ABB RAPID module: P85.mod

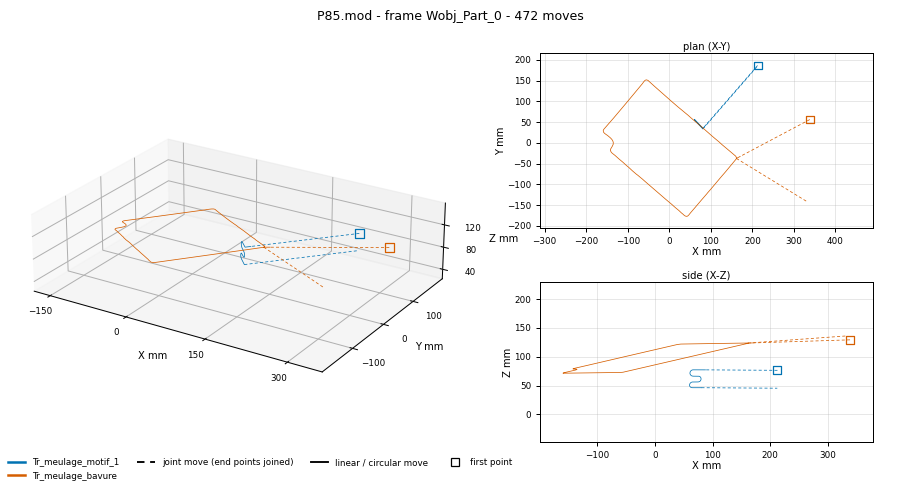
[picture p0: tool path of P85.mod in frame Wobj_Part_0, 472 of 479 moves have a stored position in this frame; points joined in program order, loops and branches not executed]
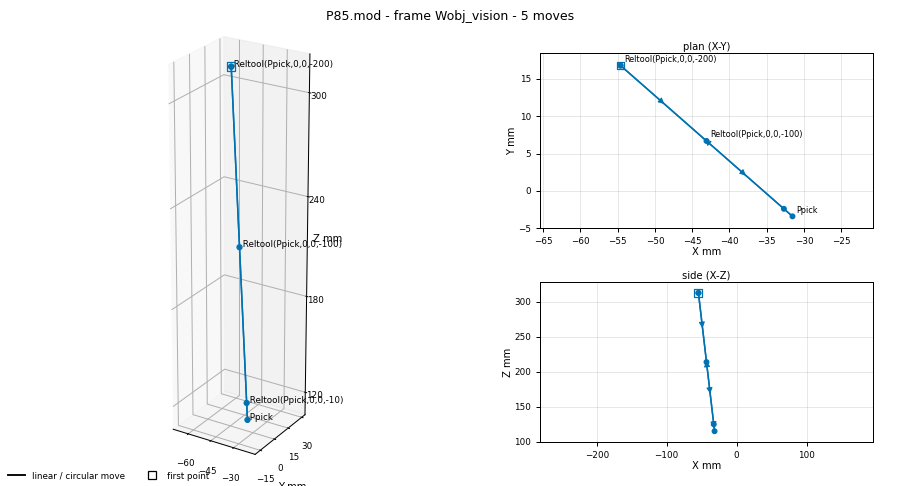
[picture p1: tool path of P85.mod in frame Wobj_vision, 5 of 479 moves have a stored position in this frame; points joined in program order, loops and branches not executed]
MODULE P85
	LOCAL CONST Speeddata vitesse_Tronconnage :=[10, 500, 0, 0];
	LOCAL CONST Robtarget Tr_meulage_motif_1_App1 :=[[212.414841209805,186.150509126283,76.4688798702914],[0.248270770432822,-0.247228008216849,-0.660888683117367,0.663676189891738],[0,0,0,0],[8.999999E+09,8.999999E+09,8.999999E+09,8.999999E+09,8.999999E+09,8.999999E+09]];
	LOCAL CONST Robtarget Tr_meulage_motif_1_App2 :=[[87.7145408886153,42.8006029953767,77.2685748528896],[0.248270770432822,-0.247228008216849,-0.660888683117367,0.663676189891738],[0,0,0,0],[8.999999E+09,8.999999E+09,8.999999E+09,8.999999E+09,8.999999E+09,8.999999E+09]];
	LOCAL CONST Robtarget Tr_meulage_motif_1_P0 :=[[81.1513671875,35.25587109375,77.3106640625],[0.248270770432822,-0.247228008216849,-0.660888683117367,0.663676189891738],[0,0,0,0],[8.999999E+09,8.999999E+09,8.999999E+09,8.999999E+09,8.999999E+09,8.999999E+09]];
	LOCAL CONST Robtarget Tr_meulage_motif_1_P1 :=[[80.4589453125,35.97736328125,77.3106875],[0.248270770432822,-0.247228008216849,-0.660888683117367,0.663676189891738],[0,0,0,0],[8.999999E+09,8.999999E+09,8.999999E+09,8.999999E+09,8.999999E+09,8.999999E+09]];
	LOCAL CONST Robtarget Tr_meulage_motif_1_P2 :=[[79.7665234375,36.69885546875,77.310703125],[0.248270770432822,-0.247228008216849,-0.660888683117367,0.663676189891738],[0,0,0,0],[8.999999E+09,8.999999E+09,8.999999E+09,8.999999E+09,8.999999E+09,8.999999E+09]];
	LOCAL CONST Robtarget Tr_meulage_motif_1_P3 :=[[79.0741015625,37.4203515625,77.3107265625],[0.248270770432822,-0.247228008216849,-0.660888683117367,0.663676189891738],[0,0,0,0],[8.999999E+09,8.999999E+09,8.999999E+09,8.999999E+09,8.999999E+09,8.999999E+09]];
	LOCAL CONST Robtarget Tr_meulage_motif_1_P4 :=[[78.3816796875,38.14184375,77.3107421875],[0.248270770432822,-0.247228008216849,-0.660888683117367,0.663676189891738],[0,0,0,0],[8.999999E+09,8.999999E+09,8.999999E+09,8.999999E+09,8.999999E+09,8.999999E+09]];
	LOCAL CONST Robtarget Tr_meulage_motif_1_P5 :=[[77.6892578125,38.8633359375,77.3107578125],[0.248270770432822,-0.247228008216849,-0.660888683117367,0.663676189891738],[0,0,0,0],[8.999999E+09,8.999999E+09,8.999999E+09,8.999999E+09,8.999999E+09,8.999999E+09]];
	LOCAL CONST Robtarget Tr_meulage_motif_1_P6 :=[[76.9968359375,39.584828125,77.31078125],[0.248270770432822,-0.247228008216849,-0.660888683117367,0.663676189891738],[0,0,0,0],[8.999999E+09,8.999999E+09,8.999999E+09,8.999999E+09,8.999999E+09,8.999999E+09]];
	LOCAL CONST Robtarget Tr_meulage_motif_1_P7 :=[[76.3044140625,40.3063203125,77.310796875],[0.248270770432822,-0.247228008216849,-0.660888683117367,0.663676189891738],[0,0,0,0],[8.999999E+09,8.999999E+09,8.999999E+09,8.999999E+09,8.999999E+09,8.999999E+09]];
	LOCAL CONST Robtarget Tr_meulage_motif_1_P8 :=[[75.6119921875,41.0278125,77.3108203125],[0.248270770432822,-0.247228008216849,-0.660888683117367,0.663676189891738],[0,0,0,0],[8.999999E+09,8.999999E+09,8.999999E+09,8.999999E+09,8.999999E+09,8.999999E+09]];
	LOCAL CONST Robtarget Tr_meulage_motif_1_P9 :=[[74.9195703125,41.7493046875,77.3108359375],[0.248270770432822,-0.247228008216849,-0.660888683117367,0.663676189891738],[0,0,0,0],[8.999999E+09,8.999999E+09,8.999999E+09,8.999999E+09,8.999999E+09,8.999999E+09]];
	LOCAL CONST Robtarget Tr_meulage_motif_1_P10 :=[[74.2271484375,42.47080078125,77.310859375],[0.248270770432822,-0.247228008216849,-0.660888683117367,0.663676189891738],[0,0,0,0],[8.999999E+09,8.999999E+09,8.999999E+09,8.999999E+09,8.999999E+09,8.999999E+09]];
	LOCAL CONST Robtarget Tr_meulage_motif_1_P11 :=[[73.5347265625,43.19229296875,77.310875],[0.248270770432822,-0.247228008216849,-0.660888683117367,0.663676189891738],[0,0,0,0],[8.999999E+09,8.999999E+09,8.999999E+09,8.999999E+09,8.999999E+09,8.999999E+09]];
	LOCAL CONST Robtarget Tr_meulage_motif_1_P12 :=[[72.8423046875,43.91378515625,77.310890625],[0.248270770432822,-0.247228008216849,-0.660888683117367,0.663676189891738],[0,0,0,0],[8.999999E+09,8.999999E+09,8.999999E+09,8.999999E+09,8.999999E+09,8.999999E+09]];
	LOCAL CONST Robtarget Tr_meulage_motif_1_P13 :=[[72.1498828125,44.63527734375,77.3109140625],[0.248270770432822,-0.247228008216849,-0.660888683117367,0.663676189891738],[0,0,0,0],[8.999999E+09,8.999999E+09,8.999999E+09,8.999999E+09,8.999999E+09,8.999999E+09]];
	LOCAL CONST Robtarget Tr_meulage_motif_1_P14 :=[[71.4574609375,45.35676953125,77.3109296875],[0.248270770432822,-0.247228008216849,-0.660888683117367,0.663676189891738],[0,0,0,0],[8.999999E+09,8.999999E+09,8.999999E+09,8.999999E+09,8.999999E+09,8.999999E+09]];
	LOCAL CONST Robtarget Tr_meulage_motif_1_P15 :=[[70.7650390625,46.07826171875,77.310953125],[0.248270770432822,-0.247228008216849,-0.660888683117367,0.663676189891738],[0,0,0,0],[8.999999E+09,8.999999E+09,8.999999E+09,8.999999E+09,8.999999E+09,8.999999E+09]];
	LOCAL CONST Robtarget Tr_meulage_motif_1_P16 :=[[70.0726171875,46.79975390625,77.31096875],[0.248270770432822,-0.247228008216849,-0.660888683117367,0.663676189891738],[0,0,0,0],[8.999999E+09,8.999999E+09,8.999999E+09,8.999999E+09,8.999999E+09,8.999999E+09]];
	LOCAL CONST Robtarget Tr_meulage_motif_1_P17 :=[[69.3801953125,47.52125,77.310984375],[0.248270770432822,-0.247228008216849,-0.660888683117367,0.663676189891738],[0,0,0,0],[8.999999E+09,8.999999E+09,8.999999E+09,8.999999E+09,8.999999E+09,8.999999E+09]];
	LOCAL CONST Robtarget Tr_meulage_motif_1_P18 :=[[68.6877734375,48.2427421875,77.3110078125],[0.248270770432822,-0.247228008216849,-0.660888683117367,0.663676189891738],[0,0,0,0],[8.999999E+09,8.999999E+09,8.999999E+09,8.999999E+09,8.999999E+09,8.999999E+09]];
	LOCAL CONST Robtarget Tr_meulage_motif_1_P19 :=[[67.9953515625,48.964234375,77.3110234375],[0.248270770432822,-0.247228008216849,-0.660888683117367,0.663676189891738],[0,0,0,0],[8.999999E+09,8.999999E+09,8.999999E+09,8.999999E+09,8.999999E+09,8.999999E+09]];
	LOCAL CONST Robtarget Tr_meulage_motif_1_P20 :=[[67.3029296875,49.6857265625,77.311046875],[0.248270770432822,-0.247228008216849,-0.660888683117367,0.663676189891738],[0,0,0,0],[8.999999E+09,8.999999E+09,8.999999E+09,8.999999E+09,8.999999E+09,8.999999E+09]];
	LOCAL CONST Robtarget Tr_meulage_motif_1_P21 :=[[66.6105078125,50.40721875,77.3110625],[0.248270770432822,-0.247228008216849,-0.660888683117367,0.663676189891738],[0,0,0,0],[8.999999E+09,8.999999E+09,8.999999E+09,8.999999E+09,8.999999E+09,8.999999E+09]];
	LOCAL CONST Robtarget Tr_meulage_motif_1_P22 :=[[65.9180859375,51.1287109375,77.3110859375],[0.248270770432822,-0.247228008216849,-0.660888683117367,0.663676189891738],[0,0,0,0],[8.999999E+09,8.999999E+09,8.999999E+09,8.999999E+09,8.999999E+09,8.999999E+09]];
	LOCAL CONST Robtarget Tr_meulage_motif_1_P23 :=[[65.22724609375,51.84141796875,77.2006171875],[0.248270770432822,-0.247228008216849,-0.660888683117367,0.663676189891738],[0,0,0,0],[8.999999E+09,8.999999E+09,8.999999E+09,8.999999E+09,8.999999E+09,8.999999E+09]];
	LOCAL CONST Robtarget Tr_meulage_motif_1_P24 :=[[64.56505859375,52.51778515625,76.98965625],[0.248270770432822,-0.247228008216849,-0.660888683117367,0.663676189891738],[0,0,0,0],[8.999999E+09,8.999999E+09,8.999999E+09,8.999999E+09,8.999999E+09,8.999999E+09]];
	LOCAL CONST Robtarget Tr_meulage_motif_1_P25 :=[[63.96585546875,53.124609375,76.7181015625],[0.248270770432822,-0.247228008216849,-0.660888683117367,0.663676189891738],[0,0,0,0],[8.999999E+09,8.999999E+09,8.999999E+09,8.999999E+09,8.999999E+09,8.999999E+09]];
	LOCAL CONST Robtarget Tr_meulage_motif_1_P26 :=[[63.43768359375,53.65715234375,76.442453125],[0.248270770432822,-0.247228008216849,-0.660888683117367,0.663676189891738],[0,0,0,0],[8.999999E+09,8.999999E+09,8.999999E+09,8.999999E+09,8.999999E+09,8.999999E+09]];
	LOCAL CONST Robtarget Tr_meulage_motif_1_P27 :=[[62.655421875,54.432515625,75.82696875],[0.248270770432822,-0.247228008216849,-0.660888683117367,0.663676189891738],[0,0,0,0],[8.999999E+09,8.999999E+09,8.999999E+09,8.999999E+09,8.999999E+09,8.999999E+09]];
	LOCAL CONST Robtarget Tr_meulage_motif_1_P28 :=[[61.91913671875,55.14502734375,74.980171875],[0.248270770432822,-0.247228008216849,-0.660888683117367,0.663676189891738],[0,0,0,0],[8.999999E+09,8.999999E+09,8.999999E+09,8.999999E+09,8.999999E+09,8.999999E+09]];
	LOCAL CONST Robtarget Tr_meulage_motif_1_P29 :=[[61.29919140625,55.724953125,73.9573359375],[0.248270770432822,-0.247228008216849,-0.660888683117367,0.663676189891738],[0,0,0,0],[8.999999E+09,8.999999E+09,8.999999E+09,8.999999E+09,8.999999E+09,8.999999E+09]];
	LOCAL CONST Robtarget Tr_meulage_motif_1_P30 :=[[60.9251953125,56.04264453125,72.8422734375],[0.248270770432822,-0.247228008216849,-0.660888683117367,0.663676189891738],[0,0,0,0],[8.999999E+09,8.999999E+09,8.999999E+09,8.999999E+09,8.999999E+09,8.999999E+09]];
	LOCAL CONST Robtarget Tr_meulage_motif_1_P31 :=[[60.884015625,56.04065625,72.147],[0.248270770432822,-0.247228008216849,-0.660888683117367,0.663676189891738],[0,0,0,0],[8.999999E+09,8.999999E+09,8.999999E+09,8.999999E+09,8.999999E+09,8.999999E+09]];
	LOCAL CONST Robtarget Tr_meulage_motif_1_P32 :=[[60.86269921875,56.0202109375,71.4864140625],[0.248270770432822,-0.247228008216849,-0.660888683117367,0.663676189891738],[0,0,0,0],[8.999999E+09,8.999999E+09,8.999999E+09,8.999999E+09,8.999999E+09,8.999999E+09]];
	LOCAL CONST Robtarget Tr_meulage_motif_1_P33 :=[[60.87937890625,55.9601796875,70.8259765625],[0.248270770432822,-0.247228008216849,-0.660888683117367,0.663676189891738],[0,0,0,0],[8.999999E+09,8.999999E+09,8.999999E+09,8.999999E+09,8.999999E+09,8.999999E+09]];
	LOCAL CONST Robtarget Tr_meulage_motif_1_P34 :=[[61.1888359375,55.56666015625,69.7253125],[0.248270770432822,-0.247228008216849,-0.660888683117367,0.663676189891738],[0,0,0,0],[8.999999E+09,8.999999E+09,8.999999E+09,8.999999E+09,8.999999E+09,8.999999E+09]];
	LOCAL CONST Robtarget Tr_meulage_motif_1_P35 :=[[61.74952734375,54.9174921875,68.7196796875],[0.248270770432822,-0.247228008216849,-0.660888683117367,0.663676189891738],[0,0,0,0],[8.999999E+09,8.999999E+09,8.999999E+09,8.999999E+09,8.999999E+09,8.999999E+09]];
	LOCAL CONST Robtarget Tr_meulage_motif_1_P36 :=[[62.43143359375,54.153484375,67.891609375],[0.248270770432822,-0.247228008216849,-0.660888683117367,0.663676189891738],[0,0,0,0],[8.999999E+09,8.999999E+09,8.999999E+09,8.999999E+09,8.999999E+09,8.999999E+09]];
	LOCAL CONST Robtarget Tr_meulage_motif_1_P37 :=[[62.89443359375,53.645515625,67.4962421875],[0.248270770432822,-0.247228008216849,-0.660888683117367,0.663676189891738],[0,0,0,0],[8.999999E+09,8.999999E+09,8.999999E+09,8.999999E+09,8.999999E+09,8.999999E+09]];
	LOCAL CONST Robtarget Tr_meulage_motif_1_P38 :=[[63.6806484375,52.79484375,67.0091796875],[0.248270770432822,-0.247228008216849,-0.660888683117367,0.663676189891738],[0,0,0,0],[8.999999E+09,8.999999E+09,8.999999E+09,8.999999E+09,8.999999E+09,8.999999E+09]];
	LOCAL CONST Robtarget Tr_meulage_motif_1_P39 :=[[64.25725390625,52.17699609375,66.745328125],[0.248270770432822,-0.247228008216849,-0.660888683117367,0.663676189891738],[0,0,0,0],[8.999999E+09,8.999999E+09,8.999999E+09,8.999999E+09,8.999999E+09,8.999999E+09]];
	LOCAL CONST Robtarget Tr_meulage_motif_1_P40 :=[[64.89599609375,51.4982421875,66.541046875],[0.248270770432822,-0.247228008216849,-0.660888683117367,0.663676189891738],[0,0,0,0],[8.999999E+09,8.999999E+09,8.999999E+09,8.999999E+09,8.999999E+09,8.999999E+09]];
	LOCAL CONST Robtarget Tr_meulage_motif_1_P41 :=[[65.5721484375,50.7866953125,66.432546875],[0.248270770432822,-0.247228008216849,-0.660888683117367,0.663676189891738],[0,0,0,0],[8.999999E+09,8.999999E+09,8.999999E+09,8.999999E+09,8.999999E+09,8.999999E+09]];
	LOCAL CONST Robtarget Tr_meulage_motif_1_P42 :=[[66.255859375,50.0671484375,66.3220390625],[0.248270770432822,-0.247228008216849,-0.660888683117367,0.663676189891738],[0,0,0,0],[8.999999E+09,8.999999E+09,8.999999E+09,8.999999E+09,8.999999E+09,8.999999E+09]];
	LOCAL CONST Robtarget Tr_meulage_motif_1_P43 :=[[66.94828125,49.34565625,66.3220234375],[0.248270770432822,-0.247228008216849,-0.660888683117367,0.663676189891738],[0,0,0,0],[8.999999E+09,8.999999E+09,8.999999E+09,8.999999E+09,8.999999E+09,8.999999E+09]];
	LOCAL CONST Robtarget Tr_meulage_motif_1_P44 :=[[67.640703125,48.6241640625,66.3220078125],[0.248270770432822,-0.247228008216849,-0.660888683117367,0.663676189891738],[0,0,0,0],[8.999999E+09,8.999999E+09,8.999999E+09,8.999999E+09,8.999999E+09,8.999999E+09]];
	LOCAL CONST Robtarget Tr_meulage_motif_1_P45 :=[[68.333125,47.902671875,66.321984375],[0.248270770432822,-0.247228008216849,-0.660888683117367,0.663676189891738],[0,0,0,0],[8.999999E+09,8.999999E+09,8.999999E+09,8.999999E+09,8.999999E+09,8.999999E+09]];
	LOCAL CONST Robtarget Tr_meulage_motif_1_P46 :=[[69.025546875,47.1811796875,66.32196875],[0.248270770432822,-0.247228008216849,-0.660888683117367,0.663676189891738],[0,0,0,0],[8.999999E+09,8.999999E+09,8.999999E+09,8.999999E+09,8.999999E+09,8.999999E+09]];
	LOCAL CONST Robtarget Tr_meulage_motif_1_P47 :=[[69.71796875,46.4596875,66.3219453125],[0.248270770432822,-0.247228008216849,-0.660888683117367,0.663676189891738],[0,0,0,0],[8.999999E+09,8.999999E+09,8.999999E+09,8.999999E+09,8.999999E+09,8.999999E+09]];
	LOCAL CONST Robtarget Tr_meulage_motif_1_P48 :=[[70.410390625,45.73819140625,66.3219296875],[0.248270770432822,-0.247228008216849,-0.660888683117367,0.663676189891738],[0,0,0,0],[8.999999E+09,8.999999E+09,8.999999E+09,8.999999E+09,8.999999E+09,8.999999E+09]];
	LOCAL CONST Robtarget Tr_meulage_motif_1_P49 :=[[71.1028125,45.01669921875,66.3219140625],[0.248270770432822,-0.247228008216849,-0.660888683117367,0.663676189891738],[0,0,0,0],[8.999999E+09,8.999999E+09,8.999999E+09,8.999999E+09,8.999999E+09,8.999999E+09]];
	LOCAL CONST Robtarget Tr_meulage_motif_1_P50 :=[[71.795234375,44.29520703125,66.321890625],[0.248270770432822,-0.247228008216849,-0.660888683117367,0.663676189891738],[0,0,0,0],[8.999999E+09,8.999999E+09,8.999999E+09,8.999999E+09,8.999999E+09,8.999999E+09]];
	LOCAL CONST Robtarget Tr_meulage_motif_1_P51 :=[[72.48765625,43.57371484375,66.321875],[0.248270770432822,-0.247228008216849,-0.660888683117367,0.663676189891738],[0,0,0,0],[8.999999E+09,8.999999E+09,8.999999E+09,8.999999E+09,8.999999E+09,8.999999E+09]];
	LOCAL CONST Robtarget Tr_meulage_motif_1_P52 :=[[73.180078125,42.85222265625,66.3218515625],[0.248270770432822,-0.247228008216849,-0.660888683117367,0.663676189891738],[0,0,0,0],[8.999999E+09,8.999999E+09,8.999999E+09,8.999999E+09,8.999999E+09,8.999999E+09]];
	LOCAL CONST Robtarget Tr_meulage_motif_1_P53 :=[[73.8725,42.13073046875,66.3218359375],[0.248270770432822,-0.247228008216849,-0.660888683117367,0.663676189891738],[0,0,0,0],[8.999999E+09,8.999999E+09,8.999999E+09,8.999999E+09,8.999999E+09,8.999999E+09]];
	LOCAL CONST Robtarget Tr_meulage_motif_1_P54 :=[[74.564921875,41.40923828125,66.3218125],[0.248270770432822,-0.247228008216849,-0.660888683117367,0.663676189891738],[0,0,0,0],[8.999999E+09,8.999999E+09,8.999999E+09,8.999999E+09,8.999999E+09,8.999999E+09]];
	LOCAL CONST Robtarget Tr_meulage_motif_1_P55 :=[[75.25734375,40.6877421875,66.321796875],[0.248270770432822,-0.247228008216849,-0.660888683117367,0.663676189891738],[0,0,0,0],[8.999999E+09,8.999999E+09,8.999999E+09,8.999999E+09,8.999999E+09,8.999999E+09]];
	LOCAL CONST Robtarget Tr_meulage_motif_1_P56 :=[[75.949765625,39.96625,66.32178125],[0.248270770432822,-0.247228008216849,-0.660888683117367,0.663676189891738],[0,0,0,0],[8.999999E+09,8.999999E+09,8.999999E+09,8.999999E+09,8.999999E+09,8.999999E+09]];
	LOCAL CONST Robtarget Tr_meulage_motif_1_P57 :=[[76.63346875,39.24670703125,66.2112734375],[0.248270770432822,-0.247228008216849,-0.660888683117367,0.663676189891738],[0,0,0,0],[8.999999E+09,8.999999E+09,8.999999E+09,8.999999E+09,8.999999E+09,8.999999E+09]];
	LOCAL CONST Robtarget Tr_meulage_motif_1_P58 :=[[77.2820390625,38.55728515625,66.00028125],[0.248270770432822,-0.247228008216849,-0.660888683117367,0.663676189891738],[0,0,0,0],[8.999999E+09,8.999999E+09,8.999999E+09,8.999999E+09,8.999999E+09,8.999999E+09]];
	LOCAL CONST Robtarget Tr_meulage_motif_1_P59 :=[[77.86371875,37.9336484375,65.7286953125],[0.248270770432822,-0.247228008216849,-0.660888683117367,0.663676189891738],[0,0,0,0],[8.999999E+09,8.999999E+09,8.999999E+09,8.999999E+09,8.999999E+09,8.999999E+09]];
	LOCAL CONST Robtarget Tr_meulage_motif_1_P60 :=[[78.3465703125,37.41090234375,65.424828125],[0.248270770432822,-0.247228008216849,-0.660888683117367,0.663676189891738],[0,0,0,0],[8.999999E+09,8.999999E+09,8.999999E+09,8.999999E+09,8.999999E+09,8.999999E+09]];
	LOCAL CONST Robtarget Tr_meulage_motif_1_P61 :=[[79.0415,36.64405859375,64.7629375],[0.248270770432822,-0.247228008216849,-0.660888683117367,0.663676189891738],[0,0,0,0],[8.999999E+09,8.999999E+09,8.999999E+09,8.999999E+09,8.999999E+09,8.999999E+09]];
	LOCAL CONST Robtarget Tr_meulage_motif_1_P62 :=[[79.6369375,35.96543359375,63.8618828125],[0.248270770432822,-0.247228008216849,-0.660888683117367,0.663676189891738],[0,0,0,0],[8.999999E+09,8.999999E+09,8.999999E+09,8.999999E+09,8.999999E+09,8.999999E+09]];
	LOCAL CONST Robtarget Tr_meulage_motif_1_P63 :=[[79.973640625,35.54712109375,62.81688671875],[0.248270770432822,-0.247228008216849,-0.660888683117367,0.663676189891738],[0,0,0,0],[8.999999E+09,8.999999E+09,8.999999E+09,8.999999E+09,8.999999E+09,8.999999E+09]];
	LOCAL CONST Robtarget Tr_meulage_motif_1_P64 :=[[80.079234375,35.39237109375,62.12435546875],[0.248270770432822,-0.247228008216849,-0.660888683117367,0.663676189891738],[0,0,0,0],[8.999999E+09,8.999999E+09,8.999999E+09,8.999999E+09,8.999999E+09,8.999999E+09]];
	LOCAL CONST Robtarget Tr_meulage_motif_1_P65 :=[[80.0986171875,35.32250390625,61.35512109375],[0.248270770432822,-0.247228008216849,-0.660888683117367,0.663676189891738],[0,0,0,0],[8.999999E+09,8.999999E+09,8.999999E+09,8.999999E+09,8.999999E+09,8.999999E+09]];
	LOCAL CONST Robtarget Tr_meulage_motif_1_P66 :=[[80.0274453125,35.34699609375,60.586015625],[0.248270770432822,-0.247228008216849,-0.660888683117367,0.663676189891738],[0,0,0,0],[8.999999E+09,8.999999E+09,8.999999E+09,8.999999E+09,8.999999E+09,8.999999E+09]];
	LOCAL CONST Robtarget Tr_meulage_motif_1_P67 :=[[79.7011796875,35.61546875,59.4788828125],[0.248270770432822,-0.247228008216849,-0.660888683117367,0.663676189891738],[0,0,0,0],[8.999999E+09,8.999999E+09,8.999999E+09,8.999999E+09,8.999999E+09,8.999999E+09]];
	LOCAL CONST Robtarget Tr_meulage_motif_1_P68 :=[[79.395421875,35.89628515625,58.89378515625],[0.248270770432822,-0.247228008216849,-0.660888683117367,0.663676189891738],[0,0,0,0],[8.999999E+09,8.999999E+09,8.999999E+09,8.999999E+09,8.999999E+09,8.999999E+09]];
	LOCAL CONST Robtarget Tr_meulage_motif_1_P69 :=[[78.7525546875,36.5089140625,58.0075625],[0.248270770432822,-0.247228008216849,-0.660888683117367,0.663676189891738],[0,0,0,0],[8.999999E+09,8.999999E+09,8.999999E+09,8.999999E+09,8.999999E+09,8.999999E+09]];
	LOCAL CONST Robtarget Tr_meulage_motif_1_P70 :=[[78.3336484375,36.91867578125,57.59367578125],[0.248270770432822,-0.247228008216849,-0.660888683117367,0.663676189891738],[0,0,0,0],[8.999999E+09,8.999999E+09,8.999999E+09,8.999999E+09,8.999999E+09,8.999999E+09]];
	LOCAL CONST Robtarget Tr_meulage_motif_1_P71 :=[[77.542046875,37.7084140625,57.05014453125],[0.248270770432822,-0.247228008216849,-0.660888683117367,0.663676189891738],[0,0,0,0],[8.999999E+09,8.999999E+09,8.999999E+09,8.999999E+09,8.999999E+09,8.999999E+09]];
	LOCAL CONST Robtarget Tr_meulage_motif_1_P72 :=[[76.960859375,38.2949375,56.75495703125],[0.248270770432822,-0.247228008216849,-0.660888683117367,0.663676189891738],[0,0,0,0],[8.999999E+09,8.999999E+09,8.999999E+09,8.999999E+09,8.999999E+09,8.999999E+09]];
	LOCAL CONST Robtarget Tr_meulage_motif_1_P73 :=[[76.3089296875,38.961046875,56.5507109375],[0.248270770432822,-0.247228008216849,-0.660888683117367,0.663676189891738],[0,0,0,0],[8.999999E+09,8.999999E+09,8.999999E+09,8.999999E+09,8.999999E+09,8.999999E+09]];
	LOCAL CONST Robtarget Tr_meulage_motif_1_P74 :=[[75.6257734375,39.6658828125,56.4422421875],[0.248270770432822,-0.247228008216849,-0.660888683117367,0.663676189891738],[0,0,0,0],[8.999999E+09,8.999999E+09,8.999999E+09,8.999999E+09,8.999999E+09,8.999999E+09]];
	LOCAL CONST Robtarget Tr_meulage_motif_1_P75 :=[[74.9349375,40.37858984375,56.33177734375],[0.248270770432822,-0.247228008216849,-0.660888683117367,0.663676189891738],[0,0,0,0],[8.999999E+09,8.999999E+09,8.999999E+09,8.999999E+09,8.999999E+09,8.999999E+09]];
	LOCAL CONST Robtarget Tr_meulage_motif_1_P76 :=[[74.242515625,41.10008203125,56.331796875],[0.248270770432822,-0.247228008216849,-0.660888683117367,0.663676189891738],[0,0,0,0],[8.999999E+09,8.999999E+09,8.999999E+09,8.999999E+09,8.999999E+09,8.999999E+09]];
	LOCAL CONST Robtarget Tr_meulage_motif_1_P77 :=[[73.55009375,41.82157421875,56.33181640625],[0.248270770432822,-0.247228008216849,-0.660888683117367,0.663676189891738],[0,0,0,0],[8.999999E+09,8.999999E+09,8.999999E+09,8.999999E+09,8.999999E+09,8.999999E+09]];
	LOCAL CONST Robtarget Tr_meulage_motif_1_P78 :=[[72.857671875,42.54306640625,56.3318359375],[0.248270770432822,-0.247228008216849,-0.660888683117367,0.663676189891738],[0,0,0,0],[8.999999E+09,8.999999E+09,8.999999E+09,8.999999E+09,8.999999E+09,8.999999E+09]];
	LOCAL CONST Robtarget Tr_meulage_motif_1_P79 :=[[72.16525,43.26455859375,56.33185546875],[0.248270770432822,-0.247228008216849,-0.660888683117367,0.663676189891738],[0,0,0,0],[8.999999E+09,8.999999E+09,8.999999E+09,8.999999E+09,8.999999E+09,8.999999E+09]];
	LOCAL CONST Robtarget Tr_meulage_motif_1_P80 :=[[71.472828125,43.9860546875,56.33187109375],[0.248270770432822,-0.247228008216849,-0.660888683117367,0.663676189891738],[0,0,0,0],[8.999999E+09,8.999999E+09,8.999999E+09,8.999999E+09,8.999999E+09,8.999999E+09]];
	LOCAL CONST Robtarget Tr_meulage_motif_1_P81 :=[[70.78040625,44.707546875,56.331890625],[0.248270770432822,-0.247228008216849,-0.660888683117367,0.663676189891738],[0,0,0,0],[8.999999E+09,8.999999E+09,8.999999E+09,8.999999E+09,8.999999E+09,8.999999E+09]];
	LOCAL CONST Robtarget Tr_meulage_motif_1_P82 :=[[70.087984375,45.4290390625,56.33191015625],[0.248270770432822,-0.247228008216849,-0.660888683117367,0.663676189891738],[0,0,0,0],[8.999999E+09,8.999999E+09,8.999999E+09,8.999999E+09,8.999999E+09,8.999999E+09]];
	LOCAL CONST Robtarget Tr_meulage_motif_1_P83 :=[[69.3955625,46.15053125,56.3319296875],[0.248270770432822,-0.247228008216849,-0.660888683117367,0.663676189891738],[0,0,0,0],[8.999999E+09,8.999999E+09,8.999999E+09,8.999999E+09,8.999999E+09,8.999999E+09]];
	LOCAL CONST Robtarget Tr_meulage_motif_1_P84 :=[[68.703140625,46.8720234375,56.33194921875],[0.248270770432822,-0.247228008216849,-0.660888683117367,0.663676189891738],[0,0,0,0],[8.999999E+09,8.999999E+09,8.999999E+09,8.999999E+09,8.999999E+09,8.999999E+09]];
	LOCAL CONST Robtarget Tr_meulage_motif_1_P85 :=[[68.01071875,47.593515625,56.33196875],[0.248270770432822,-0.247228008216849,-0.660888683117367,0.663676189891738],[0,0,0,0],[8.999999E+09,8.999999E+09,8.999999E+09,8.999999E+09,8.999999E+09,8.999999E+09]];
	LOCAL CONST Robtarget Tr_meulage_motif_1_P86 :=[[67.318296875,48.3150078125,56.331984375],[0.248270770432822,-0.247228008216849,-0.660888683117367,0.663676189891738],[0,0,0,0],[8.999999E+09,8.999999E+09,8.999999E+09,8.999999E+09,8.999999E+09,8.999999E+09]];
	LOCAL CONST Robtarget Tr_meulage_motif_1_P87 :=[[66.625875,49.03650390625,56.33200390625],[0.248270770432822,-0.247228008216849,-0.660888683117367,0.663676189891738],[0,0,0,0],[8.999999E+09,8.999999E+09,8.999999E+09,8.999999E+09,8.999999E+09,8.999999E+09]];
	LOCAL CONST Robtarget Tr_meulage_motif_1_P88 :=[[65.933453125,49.75799609375,56.3320234375],[0.248270770432822,-0.247228008216849,-0.660888683117367,0.663676189891738],[0,0,0,0],[8.999999E+09,8.999999E+09,8.999999E+09,8.999999E+09,8.999999E+09,8.999999E+09]];
	LOCAL CONST Robtarget Tr_meulage_motif_1_P89 :=[[65.24102734375,50.47948828125,56.33204296875],[0.248270770432822,-0.247228008216849,-0.660888683117367,0.663676189891738],[0,0,0,0],[8.999999E+09,8.999999E+09,8.999999E+09,8.999999E+09,8.999999E+09,8.999999E+09]];
	LOCAL CONST Robtarget Tr_meulage_motif_1_P90 :=[[64.55019140625,51.1921953125,56.221578125],[0.248270770432822,-0.247228008216849,-0.660888683117367,0.663676189891738],[0,0,0,0],[8.999999E+09,8.999999E+09,8.999999E+09,8.999999E+09,8.999999E+09,8.999999E+09]];
	LOCAL CONST Robtarget Tr_meulage_motif_1_P91 :=[[63.88800390625,51.86855859375,56.01062109375],[0.248270770432822,-0.247228008216849,-0.660888683117367,0.663676189891738],[0,0,0,0],[8.999999E+09,8.999999E+09,8.999999E+09,8.999999E+09,8.999999E+09,8.999999E+09]];
	LOCAL CONST Robtarget Tr_meulage_motif_1_P92 :=[[63.28880078125,52.47538671875,55.7390625],[0.248270770432822,-0.247228008216849,-0.660888683117367,0.663676189891738],[0,0,0,0],[8.999999E+09,8.999999E+09,8.999999E+09,8.999999E+09,8.999999E+09,8.999999E+09]];
	LOCAL CONST Robtarget Tr_meulage_motif_1_P93 :=[[62.76062890625,53.0079296875,55.4634140625],[0.248270770432822,-0.247228008216849,-0.660888683117367,0.663676189891738],[0,0,0,0],[8.999999E+09,8.999999E+09,8.999999E+09,8.999999E+09,8.999999E+09,8.999999E+09]];
	LOCAL CONST Robtarget Tr_meulage_motif_1_P94 :=[[61.9783671875,53.7832890625,54.84792578125],[0.248270770432822,-0.247228008216849,-0.660888683117367,0.663676189891738],[0,0,0,0],[8.999999E+09,8.999999E+09,8.999999E+09,8.999999E+09,8.999999E+09,8.999999E+09]];
	LOCAL CONST Robtarget Tr_meulage_motif_1_P95 :=[[61.24208203125,54.49580078125,54.00113671875],[0.248270770432822,-0.247228008216849,-0.660888683117367,0.663676189891738],[0,0,0,0],[8.999999E+09,8.999999E+09,8.999999E+09,8.999999E+09,8.999999E+09,8.999999E+09]];
	LOCAL CONST Robtarget Tr_meulage_motif_1_P96 :=[[60.62213671875,55.0757265625,52.978296875],[0.248270770432822,-0.247228008216849,-0.660888683117367,0.663676189891738],[0,0,0,0],[8.999999E+09,8.999999E+09,8.999999E+09,8.999999E+09,8.999999E+09,8.999999E+09]];
	LOCAL CONST Robtarget Tr_meulage_motif_1_P97 :=[[60.248140625,55.393421875,51.863234375],[0.248270770432822,-0.247228008216849,-0.660888683117367,0.663676189891738],[0,0,0,0],[8.999999E+09,8.999999E+09,8.999999E+09,8.999999E+09,8.999999E+09,8.999999E+09]];
	LOCAL CONST Robtarget Tr_meulage_motif_1_P98 :=[[60.2069609375,55.3914296875,51.1679609375],[0.248270770432822,-0.247228008216849,-0.660888683117367,0.663676189891738],[0,0,0,0],[8.999999E+09,8.999999E+09,8.999999E+09,8.999999E+09,8.999999E+09,8.999999E+09]];
	LOCAL CONST Robtarget Tr_meulage_motif_1_P99 :=[[60.2005703125,55.35469140625,50.4959140625],[0.248270770432822,-0.247228008216849,-0.660888683117367,0.663676189891738],[0,0,0,0],[8.999999E+09,8.999999E+09,8.999999E+09,8.999999E+09,8.999999E+09,8.999999E+09]];
	LOCAL CONST Robtarget Tr_meulage_motif_1_P100 :=[[60.22237109375,55.29264453125,49.88680078125],[0.248270770432822,-0.247228008216849,-0.660888683117367,0.663676189891738],[0,0,0,0],[8.999999E+09,8.999999E+09,8.999999E+09,8.999999E+09,8.999999E+09,8.999999E+09]];
	LOCAL CONST Robtarget Tr_meulage_motif_1_P101 :=[[60.56788671875,54.86641796875,48.86153515625],[0.248270770432822,-0.247228008216849,-0.660888683117367,0.663676189891738],[0,0,0,0],[8.999999E+09,8.999999E+09,8.999999E+09,8.999999E+09,8.999999E+09,8.999999E+09]];
	LOCAL CONST Robtarget Tr_meulage_motif_1_P102 :=[[61.167625,54.1846796875,47.98161328125],[0.248270770432822,-0.247228008216849,-0.660888683117367,0.663676189891738],[0,0,0,0],[8.999999E+09,8.999999E+09,8.999999E+09,8.999999E+09,8.999999E+09,8.999999E+09]];
	LOCAL CONST Robtarget Tr_meulage_motif_1_P103 :=[[61.577859375,53.7299375,47.55908984375],[0.248270770432822,-0.247228008216849,-0.660888683117367,0.663676189891738],[0,0,0,0],[8.999999E+09,8.999999E+09,8.999999E+09,8.999999E+09,8.999999E+09,8.999999E+09]];
	LOCAL CONST Robtarget Tr_meulage_motif_1_P104 :=[[62.3434140625,52.89802734375,47.02916015625],[0.248270770432822,-0.247228008216849,-0.660888683117367,0.663676189891738],[0,0,0,0],[8.999999E+09,8.999999E+09,8.999999E+09,8.999999E+09,8.999999E+09,8.999999E+09]];
	LOCAL CONST Robtarget Tr_meulage_motif_1_P105 :=[[62.920015625,52.2801796875,46.7653125],[0.248270770432822,-0.247228008216849,-0.660888683117367,0.663676189891738],[0,0,0,0],[8.999999E+09,8.999999E+09,8.999999E+09,8.999999E+09,8.999999E+09,8.999999E+09]];
	LOCAL CONST Robtarget Tr_meulage_motif_1_P106 :=[[63.55876171875,51.60142578125,46.56103125],[0.248270770432822,-0.247228008216849,-0.660888683117367,0.663676189891738],[0,0,0,0],[8.999999E+09,8.999999E+09,8.999999E+09,8.999999E+09,8.999999E+09,8.999999E+09]];
	LOCAL CONST Robtarget Tr_meulage_motif_1_P107 :=[[64.2349140625,50.88987890625,46.45252734375],[0.248270770432822,-0.247228008216849,-0.660888683117367,0.663676189891738],[0,0,0,0],[8.999999E+09,8.999999E+09,8.999999E+09,8.999999E+09,8.999999E+09,8.999999E+09]];
	LOCAL CONST Robtarget Tr_meulage_motif_1_P108 :=[[64.91862109375,50.17033203125,46.3420234375],[0.248270770432822,-0.247228008216849,-0.660888683117367,0.663676189891738],[0,0,0,0],[8.999999E+09,8.999999E+09,8.999999E+09,8.999999E+09,8.999999E+09,8.999999E+09]];
	LOCAL CONST Robtarget Tr_meulage_motif_1_P109 :=[[65.611046875,49.44883984375,46.34200390625],[0.248270770432822,-0.247228008216849,-0.660888683117367,0.663676189891738],[0,0,0,0],[8.999999E+09,8.999999E+09,8.999999E+09,8.999999E+09,8.999999E+09,8.999999E+09]];
	LOCAL CONST Robtarget Tr_meulage_motif_1_P110 :=[[66.30346875,48.72734765625,46.341984375],[0.248270770432822,-0.247228008216849,-0.660888683117367,0.663676189891738],[0,0,0,0],[8.999999E+09,8.999999E+09,8.999999E+09,8.999999E+09,8.999999E+09,8.999999E+09]];
	LOCAL CONST Robtarget Tr_meulage_motif_1_P111 :=[[66.995890625,48.00585546875,46.34196875],[0.248270770432822,-0.247228008216849,-0.660888683117367,0.663676189891738],[0,0,0,0],[8.999999E+09,8.999999E+09,8.999999E+09,8.999999E+09,8.999999E+09,8.999999E+09]];
	LOCAL CONST Robtarget Tr_meulage_motif_1_P112 :=[[67.6883125,47.28436328125,46.34194921875],[0.248270770432822,-0.247228008216849,-0.660888683117367,0.663676189891738],[0,0,0,0],[8.999999E+09,8.999999E+09,8.999999E+09,8.999999E+09,8.999999E+09,8.999999E+09]];
	LOCAL CONST Robtarget Tr_meulage_motif_1_P113 :=[[68.380734375,46.56287109375,46.3419296875],[0.248270770432822,-0.247228008216849,-0.660888683117367,0.663676189891738],[0,0,0,0],[8.999999E+09,8.999999E+09,8.999999E+09,8.999999E+09,8.999999E+09,8.999999E+09]];
	LOCAL CONST Robtarget Tr_meulage_motif_1_P114 :=[[69.07315625,45.841375,46.34191015625],[0.248270770432822,-0.247228008216849,-0.660888683117367,0.663676189891738],[0,0,0,0],[8.999999E+09,8.999999E+09,8.999999E+09,8.999999E+09,8.999999E+09,8.999999E+09]];
	LOCAL CONST Robtarget Tr_meulage_motif_1_P115 :=[[69.765578125,45.1198828125,46.341890625],[0.248270770432822,-0.247228008216849,-0.660888683117367,0.663676189891738],[0,0,0,0],[8.999999E+09,8.999999E+09,8.999999E+09,8.999999E+09,8.999999E+09,8.999999E+09]];
	LOCAL CONST Robtarget Tr_meulage_motif_1_P116 :=[[70.458,44.398390625,46.34187109375],[0.248270770432822,-0.247228008216849,-0.660888683117367,0.663676189891738],[0,0,0,0],[8.999999E+09,8.999999E+09,8.999999E+09,8.999999E+09,8.999999E+09,8.999999E+09]];
	LOCAL CONST Robtarget Tr_meulage_motif_1_P117 :=[[71.150421875,43.6768984375,46.34185546875],[0.248270770432822,-0.247228008216849,-0.660888683117367,0.663676189891738],[0,0,0,0],[8.999999E+09,8.999999E+09,8.999999E+09,8.999999E+09,8.999999E+09,8.999999E+09]];
	LOCAL CONST Robtarget Tr_meulage_motif_1_P118 :=[[71.84284375,42.95540625,46.3418359375],[0.248270770432822,-0.247228008216849,-0.660888683117367,0.663676189891738],[0,0,0,0],[8.999999E+09,8.999999E+09,8.999999E+09,8.999999E+09,8.999999E+09,8.999999E+09]];
	LOCAL CONST Robtarget Tr_meulage_motif_1_P119 :=[[72.535265625,42.2339140625,46.34181640625],[0.248270770432822,-0.247228008216849,-0.660888683117367,0.663676189891738],[0,0,0,0],[8.999999E+09,8.999999E+09,8.999999E+09,8.999999E+09,8.999999E+09,8.999999E+09]];
	LOCAL CONST Robtarget Tr_meulage_motif_1_P120 :=[[73.2276875,41.512421875,46.341796875],[0.248270770432822,-0.247228008216849,-0.660888683117367,0.663676189891738],[0,0,0,0],[8.999999E+09,8.999999E+09,8.999999E+09,8.999999E+09,8.999999E+09,8.999999E+09]];
	LOCAL CONST Robtarget Tr_meulage_motif_1_P121 :=[[73.920109375,40.79092578125,46.34177734375],[0.248270770432822,-0.247228008216849,-0.660888683117367,0.663676189891738],[0,0,0,0],[8.999999E+09,8.999999E+09,8.999999E+09,8.999999E+09,8.999999E+09,8.999999E+09]];
	LOCAL CONST Robtarget Tr_meulage_motif_1_P122 :=[[74.61253125,40.06943359375,46.3417578125],[0.248270770432822,-0.247228008216849,-0.660888683117367,0.663676189891738],[0,0,0,0],[8.999999E+09,8.999999E+09,8.999999E+09,8.999999E+09,8.999999E+09,8.999999E+09]];
	LOCAL CONST Robtarget Tr_meulage_motif_1_P123 :=[[75.304953125,39.34794140625,46.3417421875],[0.248270770432822,-0.247228008216849,-0.660888683117367,0.663676189891738],[0,0,0,0],[8.999999E+09,8.999999E+09,8.999999E+09,8.999999E+09,8.999999E+09,8.999999E+09]];
	LOCAL CONST Robtarget Tr_meulage_motif_1_P124 :=[[75.997375,38.62644921875,46.34172265625],[0.248270770432822,-0.247228008216849,-0.660888683117367,0.663676189891738],[0,0,0,0],[8.999999E+09,8.999999E+09,8.999999E+09,8.999999E+09,8.999999E+09,8.999999E+09]];
	LOCAL CONST Robtarget Tr_meulage_motif_1_P125 :=[[76.689796875,37.90495703125,46.341703125],[0.248270770432822,-0.247228008216849,-0.660888683117367,0.663676189891738],[0,0,0,0],[8.999999E+09,8.999999E+09,8.999999E+09,8.999999E+09,8.999999E+09,8.999999E+09]];
	LOCAL CONST Robtarget Tr_meulage_motif_1_P126 :=[[77.38221875,37.18346484375,46.34168359375],[0.248270770432822,-0.247228008216849,-0.660888683117367,0.663676189891738],[0,0,0,0],[8.999999E+09,8.999999E+09,8.999999E+09,8.999999E+09,8.999999E+09,8.999999E+09]];
	LOCAL CONST Robtarget Tr_meulage_motif_1_P127 :=[[78.074640625,36.46197265625,46.3416640625],[0.248270770432822,-0.247228008216849,-0.660888683117367,0.663676189891738],[0,0,0,0],[8.999999E+09,8.999999E+09,8.999999E+09,8.999999E+09,8.999999E+09,8.999999E+09]];
	LOCAL CONST Robtarget Tr_meulage_motif_1_P128 :=[[78.7670625,35.7404765625,46.34164453125],[0.248270770432822,-0.247228008216849,-0.660888683117367,0.663676189891738],[0,0,0,0],[8.999999E+09,8.999999E+09,8.999999E+09,8.999999E+09,8.999999E+09,8.999999E+09]];
	LOCAL CONST Robtarget Tr_meulage_motif_1_P129 :=[[79.459484375,35.018984375,46.341625],[0.248270770432822,-0.247228008216849,-0.660888683117367,0.663676189891738],[0,0,0,0],[8.999999E+09,8.999999E+09,8.999999E+09,8.999999E+09,8.999999E+09,8.999999E+09]];
	LOCAL CONST Robtarget Tr_meulage_motif_1_P130 :=[[80.15190625,34.2974921875,46.341609375],[0.248270770432822,-0.247228008216849,-0.660888683117367,0.663676189891738],[0,0,0,0],[8.999999E+09,8.999999E+09,8.999999E+09,8.999999E+09,8.999999E+09,8.999999E+09]];
	LOCAL CONST Robtarget Tr_meulage_motif_1_P131 :=[[80.844328125,33.576,46.34158984375],[0.248270770432822,-0.247228008216849,-0.660888683117367,0.663676189891738],[0,0,0,0],[8.999999E+09,8.999999E+09,8.999999E+09,8.999999E+09,8.999999E+09,8.999999E+09]];
	LOCAL CONST Robtarget Tr_meulage_motif_1_degg1 :=[[87.4075018261153,41.1207319016267,46.2995006341396],[0.248270770432822,-0.247228008216849,-0.660888683117367,0.663676189891738],[0,0,0,0],[8.999999E+09,8.999999E+09,8.999999E+09,8.999999E+09,8.999999E+09,8.999999E+09]];
	LOCAL CONST Robtarget Tr_meulage_motif_1_degg2 :=[[212.107802147305,184.470638032533,45.4998056515414],[0.248270770432822,-0.247228008216849,-0.660888683117367,0.663676189891738],[0,0,0,0],[8.999999E+09,8.999999E+09,8.999999E+09,8.999999E+09,8.999999E+09,8.999999E+09]];
	LOCAL CONST Robtarget Tr_meulage_bavure_App1 :=[[338.141353099256,56.1089656824525,129.270502837446],[0.359477377125384,-0.369677564038208,-0.614267705755514,0.597318758827888],[0,0,0,0],[8.999999E+09,8.999999E+09,8.999999E+09,8.999999E+09,8.999999E+09,8.999999E+09]];
	LOCAL CONST Robtarget Tr_meulage_bavure_App2 :=[[170.321691873713,-32.8197372627524,123.955702876247],[0.359477377125384,-0.369677564038208,-0.614267705755514,0.597318758827888],[0,0,0,0],[8.999999E+09,8.999999E+09,8.999999E+09,8.999999E+09,8.999999E+09,8.999999E+09]];
	LOCAL CONST Robtarget Tr_meulage_bavure_P0 :=[[161.489078125,-37.5001953125,123.6759765625],[0.359477377125384,-0.369677564038208,-0.614267705755514,0.597318758827888],[0,0,0,0],[8.999999E+09,8.999999E+09,8.999999E+09,8.999999E+09,8.999999E+09,8.999999E+09]];
	LOCAL CONST Robtarget Tr_meulage_bavure_P1 :=[[161.82421875,-36.49319921875,123.6161953125],[0.35276726064605,-0.362677382629981,-0.618315579063414,0.601420169791822],[0,0,0,0],[8.999999E+09,8.999999E+09,8.999999E+09,8.999999E+09,8.999999E+09,8.999999E+09]];
	LOCAL CONST Robtarget Tr_meulage_bavure_P2 :=[[160.123765625,-32.58012109375,122.961890625],[0.334619948848255,-0.343734165055808,-0.628713112754664,0.612042592845073],[0,0,0,0],[8.999999E+09,8.999999E+09,8.999999E+09,8.999999E+09,8.999999E+09,8.999999E+09]];
	LOCAL CONST Robtarget Tr_meulage_bavure_P3 :=[[160.0276875,-32.218830078125,122.9100390625],[0.310221226304004,-0.318237503792412,-0.641465721515757,0.625307452418955],[0,0,0,0],[8.999999E+09,8.999999E+09,8.999999E+09,8.999999E+09,8.999999E+09,8.999999E+09]];
	LOCAL CONST Robtarget Tr_meulage_bavure_P4 :=[[159.97871875,-32.15770703125,122.896671875],[0.28573180537606,-0.29257522346814,-0.652864166250617,0.63759348681977],[0,0,0,0],[8.999999E+09,8.999999E+09,8.999999E+09,8.999999E+09,8.999999E+09,8.999999E+09]];
	LOCAL CONST Robtarget Tr_meulage_bavure_P5 :=[[157.63534375,-30.1469609375,122.3539140625],[0.265599829666162,-0.271343026137636,-0.661111066546468,0.647118111582089],[0,0,0,0],[8.999999E+09,8.999999E+09,8.999999E+09,8.999999E+09,8.999999E+09,8.999999E+09]];
	LOCAL CONST Robtarget Tr_meulage_bavure_P6 :=[[156.706078125,-29.36853515625,122.1406953125],[0.251589982396947,-0.256350873560219,-0.666075318949548,0.653705116905685],[0,0,0,0],[8.999999E+09,8.999999E+09,8.999999E+09,8.999999E+09,8.999999E+09,8.999999E+09]];
	LOCAL CONST Robtarget Tr_meulage_bavure_P7 :=[[154.6675625,-27.83671875,121.6916171875],[0.243317460991168,-0.247193173331807,-0.668428324276981,0.657948116145361],[0,0,0,0],[8.999999E+09,8.999999E+09,8.999999E+09,8.999999E+09,8.999999E+09,8.999999E+09]];
	LOCAL CONST Robtarget Tr_meulage_bavure_P8 :=[[152.40115625,-25.954478515625,121.1733203125],[0.239445955854181,-0.242488888572142,-0.66896403426586,0.66056937107534],[0,0,0,0],[8.999999E+09,8.999999E+09,8.999999E+09,8.999999E+09,8.999999E+09,8.999999E+09]];
	LOCAL CONST Robtarget Tr_meulage_bavure_P9 :=[[151.625421875,-25.30837890625,120.9957265625],[0.238504842188388,-0.240729489706835,-0.668349683828104,0.662173280316454],[0,0,0,0],[8.999999E+09,8.999999E+09,8.999999E+09,8.999999E+09,8.999999E+09,8.999999E+09]];
	LOCAL CONST Robtarget Tr_meulage_bavure_P10 :=[[150.8259375,-24.604099609375,120.808609375],[0.239215889276791,-0.240619293365567,-0.667103510284543,0.663212651073402],[0,0,0,0],[8.999999E+09,8.999999E+09,8.999999E+09,8.999999E+09,8.999999E+09,8.999999E+09]];
	LOCAL CONST Robtarget Tr_meulage_bavure_P11 :=[[148.72865625,-22.751873046875,120.317265625],[0.240678495084672,-0.241250604579521,-0.665571384524457,0.6639930269935],[0,0,0,0],[8.999999E+09,8.999999E+09,8.999999E+09,8.999999E+09,8.999999E+09,8.999999E+09]];
	LOCAL CONST Robtarget Tr_meulage_bavure_P12 :=[[147.762953125,-21.93584375,120.0949375],[0.242257324128803,-0.241994904684668,-0.66400042148895,0.664720464011082],[0,0,0,0],[8.999999E+09,8.999999E+09,8.999999E+09,8.999999E+09,8.999999E+09,8.999999E+09]];
	LOCAL CONST Robtarget Tr_meulage_bavure_P13 :=[[144.529953125,-19.1548046875,119.3453984375],[0.243613530504702,-0.242519900553449,-0.662521289825167,0.66550889259196],[0,0,0,0],[8.999999E+09,8.999999E+09,8.999999E+09,8.999999E+09,8.999999E+09,8.999999E+09]];
	LOCAL CONST Robtarget Tr_meulage_bavure_P14 :=[[140.923734375,-16.0849228515625,118.51275],[0.244583140196905,-0.242675302484408,-0.661205946901556,0.666404142302206],[0,0,0,0],[8.999999E+09,8.999999E+09,8.999999E+09,8.999999E+09,8.999999E+09,8.999999E+09]];
	LOCAL CONST Robtarget Tr_meulage_bavure_P15 :=[[140.658296875,-15.8480673828125,118.4503046875],[0.24515542713548,-0.242462567690669,-0.660067870832464,0.667398775627859],[0,0,0,0],[8.999999E+09,8.999999E+09,8.999999E+09,8.999999E+09,8.999999E+09,8.999999E+09]];
	LOCAL CONST Robtarget Tr_meulage_bavure_P16 :=[[140.569625,-15.768974609375,118.4294453125],[0.245478401979063,-0.242033825820144,-0.659055657629629,0.668435203641345],[0,0,0,0],[8.999999E+09,8.999999E+09,8.999999E+09,8.999999E+09,8.999999E+09,8.999999E+09]];
	LOCAL CONST Robtarget Tr_meulage_bavure_P17 :=[[136.065,-12.0183330078125,117.39828125],[0.245769274802604,-0.24160417173166,-0.658089681289081,0.669434731057253],[0,0,0,0],[8.999999E+09,8.999999E+09,8.999999E+09,8.999999E+09,8.999999E+09,8.999999E+09]];
	LOCAL CONST Robtarget Tr_meulage_bavure_P18 :=[[135.63234375,-11.6969228515625,117.303359375],[0.246224991679659,-0.241371389303987,-0.65710478553598,0.670318138441389],[0,0,0,0],[8.999999E+09,8.999999E+09,8.999999E+09,8.999999E+09,8.999999E+09,8.999999E+09]];
	LOCAL CONST Robtarget Tr_meulage_bavure_P19 :=[[131.931359375,-8.6471328125,116.4595234375],[0.246939345125507,-0.241430373774351,-0.656073532695082,0.671043854114735],[0,0,0,0],[8.999999E+09,8.999999E+09,8.999999E+09,8.999999E+09,8.999999E+09,8.999999E+09]];
	LOCAL CONST Robtarget Tr_meulage_bavure_P20 :=[[130.685125,-7.589390625,116.172109375],[0.247819551442662,-0.241690516836492,-0.655031986802466,0.671642955936919],[0,0,0,0],[8.999999E+09,8.999999E+09,8.999999E+09,8.999999E+09,8.999999E+09,8.999999E+09]];
	LOCAL CONST Robtarget Tr_meulage_bavure_P21 :=[[129.8374921875,-6.92769091796875,115.9827578125],[0.248623123100672,-0.241913600546654,-0.654066087893379,0.672206742898398],[0,0,0,0],[8.999999E+09,8.999999E+09,8.999999E+09,8.999999E+09,8.999999E+09,8.999999E+09]];
	LOCAL CONST Robtarget Tr_meulage_bavure_P22 :=[[126.4407734375,-3.92382104492187,115.1865546875],[0.249078840737307,-0.241841360132536,-0.653278866723014,0.672829257627296],[0,0,0,0],[8.999999E+09,8.999999E+09,8.999999E+09,8.999999E+09,8.999999E+09,8.999999E+09]];
	LOCAL CONST Robtarget Tr_meulage_bavure_P23 :=[[123.95246875,-1.51439392089844,114.5811171875],[0.249048740869028,-0.241348545497409,-0.652727199143116,0.673552379371211],[0,0,0,0],[8.999999E+09,8.999999E+09,8.999999E+09,8.999999E+09,8.999999E+09,8.999999E+09]];
	LOCAL CONST Robtarget Tr_meulage_bavure_P24 :=[[119.3564765625,2.62285107421875,113.496078125],[0.24864716519142,-0.240550377681981,-0.652371740002208,0.674330197963742],[0,0,0,0],[8.999999E+09,8.999999E+09,8.999999E+09,8.999999E+09,8.999999E+09,8.999999E+09]];
	LOCAL CONST Robtarget Tr_meulage_bavure_P25 :=[[115.885734375,5.61625048828125,112.6905859375],[0.248206292848843,-0.239770955969502,-0.652095637374118,0.675036891274357],[0,0,0,0],[8.999999E+09,8.999999E+09,8.999999E+09,8.999999E+09,8.999999E+09,8.999999E+09]];
	LOCAL CONST Robtarget Tr_meulage_bavure_P26 :=[[113.5089765625,7.601833984375,112.1458125],[0.248137564196063,-0.239409643083424,-0.651756905236743,0.675517363588632],[0,0,0,0],[8.999999E+09,8.999999E+09,8.999999E+09,8.999999E+09,8.999999E+09,8.999999E+09]];
	LOCAL CONST Robtarget Tr_meulage_bavure_P27 :=[[109.6526328125,10.6559951171875,111.279671875],[0.248714830495185,-0.23973529579508,-0.65126758705549,0.675661491497567],[0,0,0,0],[8.999999E+09,8.999999E+09,8.999999E+09,8.999999E+09,8.999999E+09,8.999999E+09]];
	LOCAL CONST Robtarget Tr_meulage_bavure_P28 :=[[107.6943828125,12.2560068359375,110.834640625],[0.249937133301145,-0.24074489144693,-0.65062651902724,0.675469066188755],[0,0,0,0],[8.999999E+09,8.999999E+09,8.999999E+09,8.999999E+09,8.999999E+09,8.999999E+09]];
	LOCAL CONST Robtarget Tr_meulage_bavure_P29 :=[[106.4360078125,13.31462890625,110.5454296875],[0.251519125482931,-0.242163107266078,-0.64993256180357,0.675042831309976],[0,0,0,0],[8.999999E+09,8.999999E+09,8.999999E+09,8.999999E+09,8.999999E+09,8.999999E+09]];
	LOCAL CONST Robtarget Tr_meulage_bavure_P30 :=[[102.2531484375,16.95091015625,109.5716171875],[0.252979423972975,-0.243526379545889,-0.649355572535836,0.674561823651643],[0,0,0,0],[8.999999E+09,8.999999E+09,8.999999E+09,8.999999E+09,8.999999E+09,8.999999E+09]];
	LOCAL CONST Robtarget Tr_meulage_bavure_P31 :=[[99.8893203125,19.05167578125,109.0164375],[0.253800967500349,-0.244336840431315,-0.64908192865146,0.674223425284252],[0,0,0,0],[8.999999E+09,8.999999E+09,8.999999E+09,8.999999E+09,8.999999E+09,8.999999E+09]];
	LOCAL CONST Robtarget Tr_meulage_bavure_P32 :=[[97.3266796875,21.390537109375,108.4080390625],[0.253529025277429,-0.24415274372284,-0.649273600872682,0.67420787764925],[0,0,0,0],[8.999999E+09,8.999999E+09,8.999999E+09,8.999999E+09,8.999999E+09,8.999999E+09]];
	LOCAL CONST Robtarget Tr_meulage_bavure_P33 :=[[93.232828125,25.031400390625,107.4462578125],[0.251810781716999,-0.242628410212318,-0.650051207005374,0.674652661033641],[0,0,0,0],[8.999999E+09,8.999999E+09,8.999999E+09,8.999999E+09,8.999999E+09,8.999999E+09]];
	LOCAL CONST Robtarget Tr_meulage_bavure_P34 :=[[93.0785859375,25.147248046875,107.41228125],[0.248462599906379,-0.239578923049632,-0.651463937504961,0.675620466096664],[0,0,0,0],[8.999999E+09,8.999999E+09,8.999999E+09,8.999999E+09,8.999999E+09,8.999999E+09]];
	LOCAL CONST Robtarget Tr_meulage_bavure_P35 :=[[92.3705546875,25.784333984375,107.24515625],[0.243518614959495,-0.235020778346356,-0.653462293903926,0.677090059267969],[0,0,0,0],[8.999999E+09,8.999999E+09,8.999999E+09,8.999999E+09,8.999999E+09,8.999999E+09]];
	LOCAL CONST Robtarget Tr_meulage_bavure_P36 :=[[87.9107421875,29.58517578125,106.2149609375],[0.237334935233677,-0.229283250470837,-0.655880266870699,0.678912656459411],[0,0,0,0],[8.999999E+09,8.999999E+09,8.999999E+09,8.999999E+09,8.999999E+09,8.999999E+09]];
	LOCAL CONST Robtarget Tr_meulage_bavure_P37 :=[[86.7107734375,30.652931640625,105.9329921875],[0.230657355959346,-0.223073230789016,-0.658428403000887,0.68081389231485],[0,0,0,0],[8.999999E+09,8.999999E+09,8.999999E+09,8.999999E+09,8.999999E+09,8.999999E+09]];
	LOCAL CONST Robtarget Tr_meulage_bavure_P38 :=[[79.018734375,37.43833984375,104.1317578125],[0.224504554009201,-0.217366062427621,-0.660757934268434,0.682457802677318],[0,0,0,0],[8.999999E+09,8.999999E+09,8.999999E+09,8.999999E+09,8.999999E+09,8.999999E+09]];
	LOCAL CONST Robtarget Tr_meulage_bavure_P39 :=[[78.4500703125,37.98322265625,103.9940078125],[0.219932132075249,-0.213176061360495,-0.66254111170384,0.683538659803453],[0,0,0,0],[8.999999E+09,8.999999E+09,8.999999E+09,8.999999E+09,8.999999E+09,8.999999E+09]];
	LOCAL CONST Robtarget Tr_meulage_bavure_P40 :=[[78.2325859375,38.116703125,103.9492734375],[0.217710439625849,-0.211245846415385,-0.663557154230322,0.683863480469548],[0,0,0,0],[8.999999E+09,8.999999E+09,8.999999E+09,8.999999E+09,8.999999E+09,8.999999E+09]];
	LOCAL CONST Robtarget Tr_meulage_bavure_P41 :=[[77.1535703125,39.03486328125,103.7001796875],[0.218079437222146,-0.211806836613365,-0.66373915622331,0.68339560689302],[0,0,0,0],[8.999999E+09,8.999999E+09,8.999999E+09,8.999999E+09,8.999999E+09,8.999999E+09]];
	LOCAL CONST Robtarget Tr_meulage_bavure_P42 :=[[69.8700625,45.0931953125,102.03353125],[0.220703950296817,-0.214533228613105,-0.663174567040075,0.682249773745237],[0,0,0,0],[8.999999E+09,8.999999E+09,8.999999E+09,8.999999E+09,8.999999E+09,8.999999E+09]];
	LOCAL CONST Robtarget Tr_meulage_bavure_P43 :=[[69.24584375,45.7311328125,101.87809375],[0.224815400426383,-0.218673925461375,-0.662069702543715,0.680663983936358],[0,0,0,0],[8.999999E+09,8.999999E+09,8.999999E+09,8.999999E+09,8.999999E+09,8.999999E+09]];
	LOCAL CONST Robtarget Tr_meulage_bavure_P44 :=[[67.346625,47.147765625,101.4608203125],[0.229502618739731,-0.223337029198313,-0.660687295502464,0.678926665363879],[0,0,0,0],[8.999999E+09,8.999999E+09,8.999999E+09,8.999999E+09,8.999999E+09,8.999999E+09]];
	LOCAL CONST Robtarget Tr_meulage_bavure_P45 :=[[64.41136328125,49.7630625,100.77071875],[0.233962084943426,-0.227734476747008,-0.659280616408619,0.677309249706191],[0,0,0,0],[8.999999E+09,8.999999E+09,8.999999E+09,8.999999E+09,8.999999E+09,8.999999E+09]];
	LOCAL CONST Robtarget Tr_meulage_bavure_P46 :=[[62.6122890625,51.225375,100.362671875],[0.237684031432284,-0.231361852349466,-0.658023809856216,0.676004926122459],[0,0,0,0],[8.999999E+09,8.999999E+09,8.999999E+09,8.999999E+09,8.999999E+09,8.999999E+09]];
	LOCAL CONST Robtarget Tr_meulage_bavure_P47 :=[[61.56168359375,52.155828125,100.1162578125],[0.240506692331351,-0.234060809601102,-0.656989646837627,0.675082715154876],[0,0,0,0],[8.999999E+09,8.999999E+09,8.999999E+09,8.999999E+09,8.999999E+09,8.999999E+09]];
	LOCAL CONST Robtarget Tr_meulage_bavure_P48 :=[[60.5981640625,53.092015625,99.881484375],[0.242536299612786,-0.235931155863053,-0.656151147146801,0.674520796685468],[0,0,0,0],[8.999999E+09,8.999999E+09,8.999999E+09,8.999999E+09,8.999999E+09,8.999999E+09]];
	LOCAL CONST Robtarget Tr_meulage_bavure_P49 :=[[59.23597265625,54.213703125,99.570984375],[0.244027987794599,-0.237223397629389,-0.655430025546311,0.674230585484262],[0,0,0,0],[8.999999E+09,8.999999E+09,8.999999E+09,8.999999E+09,8.999999E+09,8.999999E+09]];
	LOCAL CONST Robtarget Tr_meulage_bavure_P50 :=[[55.27891796875,57.5543125,98.660296875],[0.245231336685715,-0.238186154976481,-0.65474937940558,0.67411586337429],[0,0,0,0],[8.999999E+09,8.999999E+09,8.999999E+09,8.999999E+09,8.999999E+09,8.999999E+09]];
	LOCAL CONST Robtarget Tr_meulage_bavure_P51 :=[[51.732703125,60.4791484375,97.85146875],[0.246293097172888,-0.238965546335283,-0.654063154875077,0.674119104746726],[0,0,0,0],[8.999999E+09,8.999999E+09,8.999999E+09,8.999999E+09,8.999999E+09,8.999999E+09]];
	LOCAL CONST Robtarget Tr_meulage_bavure_P52 :=[[49.80992578125,62.2975625,97.3882421875],[0.247240324619471,-0.23959589900202,-0.653372346104257,0.674218513843762],[0,0,0,0],[8.999999E+09,8.999999E+09,8.999999E+09,8.999999E+09,8.999999E+09,8.999999E+09]];
	LOCAL CONST Robtarget Tr_meulage_bavure_P53 :=[[46.54223046875,65.22901953125,96.617859375],[0.248014128377632,-0.240028025281187,-0.652707726042913,0.674424320119453],[0,0,0,0],[8.999999E+09,8.999999E+09,8.999999E+09,8.999999E+09,8.999999E+09,8.999999E+09]];
	LOCAL CONST Robtarget Tr_meulage_bavure_P54 :=[[45.20770703125,66.4407265625,96.3016953125],[0.248555917969701,-0.240214860805124,-0.652101535809153,0.674744665251944],[0,0,0,0],[8.999999E+09,8.999999E+09,8.999999E+09,8.999999E+09,8.999999E+09,8.999999E+09]];
	LOCAL CONST Robtarget Tr_meulage_bavure_P55 :=[[42.898796875,68.4261875,95.76646875],[0.248857440892654,-0.240161465685204,-0.651571637584466,0.675164310081473],[0,0,0,0],[8.999999E+09,8.999999E+09,8.999999E+09,8.999999E+09,8.999999E+09,8.999999E+09]];
	LOCAL CONST Robtarget Tr_meulage_bavure_P56 :=[[41.5326171875,69.52171875,95.4581953125],[0.248953171727383,-0.239910265427149,-0.651115638702003,0.675658055429841],[0,0,0,0],[8.999999E+09,8.999999E+09,8.999999E+09,8.999999E+09,8.999999E+09,8.999999E+09]];
	LOCAL CONST Robtarget Tr_meulage_bavure_P57 :=[[37.16591796875,73.0086796875,94.4743984375],[0.248895759710229,-0.239522612371433,-0.650726645242216,0.676191283685944],[0,0,0,0],[8.999999E+09,8.999999E+09,8.999999E+09,8.999999E+09,8.999999E+09,8.999999E+09]];
	LOCAL CONST Robtarget Tr_meulage_bavure_P58 :=[[34.9973828125,74.7069296875,93.9893828125],[0.248725907822635,-0.239049436197567,-0.650403876986076,0.676731546946729],[0,0,0,0],[8.999999E+09,8.999999E+09,8.999999E+09,8.999999E+09,8.999999E+09,8.999999E+09]];
	LOCAL CONST Robtarget Tr_meulage_bavure_P59 :=[[31.93165234375,77.40484375,93.272171875],[0.248480251742954,-0.238533540376053,-0.650143357909113,0.677253961801692],[0,0,0,0],[8.999999E+09,8.999999E+09,8.999999E+09,8.999999E+09,8.999999E+09,8.999999E+09]];
	LOCAL CONST Robtarget Tr_meulage_bavure_P60 :=[[31.637072265625,77.6556875,93.2041484375],[0.248211572814999,-0.23803730960426,-0.64994108448808,0.677721064341022],[0,0,0,0],[8.999999E+09,8.999999E+09,8.999999E+09,8.999999E+09,8.999999E+09,8.999999E+09]];
	LOCAL CONST Robtarget Tr_meulage_bavure_P61 :=[[21.98300390625,85.5757734375,91.0067421875],[0.248026379412664,-0.237666602301944,-0.649764878738832,0.678087828841667],[0,0,0,0],[8.999999E+09,8.999999E+09,8.999999E+09,8.999999E+09,8.999999E+09,8.999999E+09]];
	LOCAL CONST Robtarget Tr_meulage_bavure_P62 :=[[21.499533203125,86.052828125,90.8881640625],[0.24805501730923,-0.237551844329973,-0.649576994307201,0.678297543936264],[0,0,0,0],[8.999999E+09,8.999999E+09,8.999999E+09,8.999999E+09,8.999999E+09,8.999999E+09]];
	LOCAL CONST Robtarget Tr_meulage_bavure_P63 :=[[20.596056640625,86.751,90.6870859375],[0.248407390839962,-0.237799874284377,-0.649341772610292,0.678306899795175],[0,0,0,0],[8.999999E+09,8.999999E+09,8.999999E+09,8.999999E+09,8.999999E+09,8.999999E+09]];
	LOCAL CONST Robtarget Tr_meulage_bavure_P64 :=[[15.50149609375,91.2400078125,89.494640625],[0.249123933311026,-0.238452689571482,-0.64904892172772,0.678095183504392],[0,0,0,0],[8.999999E+09,8.999999E+09,8.999999E+09,8.999999E+09,8.999999E+09,8.999999E+09]];
	LOCAL CONST Robtarget Tr_meulage_bavure_P65 :=[[13.61288671875,92.9689765625,89.045703125],[0.250160159342188,-0.239467253240438,-0.648711786666116,0.6776786459258],[0,0,0,0],[8.999999E+09,8.999999E+09,8.999999E+09,8.999999E+09,8.999999E+09,8.999999E+09]];
	LOCAL CONST Robtarget Tr_meulage_bavure_P66 :=[[8.2011005859375,97.5695859375,87.796828125],[0.251400520207656,-0.2407297972956,-0.648364585542019,0.677104354843672],[0,0,0,0],[8.999999E+09,8.999999E+09,8.999999E+09,8.999999E+09,8.999999E+09,8.999999E+09]];
	LOCAL CONST Robtarget Tr_meulage_bavure_P67 :=[[5.03517431640625,100.1880625,87.07396875],[0.25269462049887,-0.24208939073124,-0.648049774651745,0.676438944207186],[0,0,0,0],[8.999999E+09,8.999999E+09,8.999999E+09,8.999999E+09,8.999999E+09,8.999999E+09]];
	LOCAL CONST Robtarget Tr_meulage_bavure_P68 :=[[3.12470825195313,101.759484375,86.6386875],[0.253891815433018,-0.243396021665721,-0.647813013717262,0.675748194190695],[0,0,0,0],[8.999999E+09,8.999999E+09,8.999999E+09,8.999999E+09,8.999999E+09,8.999999E+09]];
	LOCAL CONST Robtarget Tr_meulage_bavure_P69 :=[[0.516263000488281,104.148734375,86.0185078125],[0.254859472441788,-0.244511797504982,-0.647689329953388,0.675099371983197],[0,0,0,0],[8.999999E+09,8.999999E+09,8.999999E+09,8.999999E+09,8.999999E+09,8.999999E+09]];
	LOCAL CONST Robtarget Tr_meulage_bavure_P70 :=[[-2.00272412109375,106.4556953125,85.4196328125],[0.255502055546817,-0.245331423494274,-0.647698580582508,0.674550028514586],[0,0,0,0],[8.999999E+09,8.999999E+09,8.999999E+09,8.999999E+09,8.999999E+09,8.999999E+09]];
	LOCAL CONST Robtarget Tr_meulage_bavure_P71 :=[[-3.32872973632813,107.582546875,85.113671875],[0.255782659378091,-0.245803134233467,-0.647836972793565,0.674138937492965],[0,0,0,0],[8.999999E+09,8.999999E+09,8.999999E+09,8.999999E+09,8.999999E+09,8.999999E+09]];
	LOCAL CONST Robtarget Tr_meulage_bavure_P72 :=[[-11.8568388671875,115.0172421875,83.1260234375],[0.255737481530467,-0.245942953439845,-0.648071031621972,0.673880065120028],[0,0,0,0],[8.999999E+09,8.999999E+09,8.999999E+09,8.999999E+09,8.999999E+09,8.999999E+09]];
	LOCAL CONST Robtarget Tr_meulage_bavure_P73 :=[[-12.4804921875,115.5860390625,82.9780078125],[0.255475044435192,-0.245837185732095,-0.648340897890752,0.673758606553099],[0,0,0,0],[8.999999E+09,8.999999E+09,8.999999E+09,8.999999E+09,8.999999E+09,8.999999E+09]];
	LOCAL CONST Robtarget Tr_meulage_bavure_P74 :=[[-22.1798984375,124.1585703125,80.704984375],[0.255164962103322,-0.245628751418856,-0.648560888039154,0.673740404827474],[0,0,0,0],[8.999999E+09,8.999999E+09,8.999999E+09,8.999999E+09,8.999999E+09,8.999999E+09]];
	LOCAL CONST Robtarget Tr_meulage_bavure_P75 :=[[-25.44776953125,127.0613984375,79.9376171875],[0.254968108910684,-0.245456157745685,-0.648652731410122,0.673789412277622],[0,0,0,0],[8.999999E+09,8.999999E+09,8.999999E+09,8.999999E+09,8.999999E+09,8.999999E+09]];
	LOCAL CONST Robtarget Tr_meulage_bavure_P76 :=[[-25.52045703125,127.120828125,79.92109375],[0.255005535816973,-0.2454157784332,-0.648548196664394,0.67389057643069],[0,0,0,0],[8.999999E+09,8.999999E+09,8.999999E+09,8.999999E+09,8.999999E+09,8.999999E+09]];
	LOCAL CONST Robtarget Tr_meulage_bavure_P77 :=[[-25.83838671875,127.390828125,79.84775],[0.255282919213362,-0.245498013400582,-0.64822749747094,0.674064142420315],[0,0,0,0],[8.999999E+09,8.999999E+09,8.999999E+09,8.999999E+09,8.999999E+09,8.999999E+09]];
	LOCAL CONST Robtarget Tr_meulage_bavure_P78 :=[[-35.36965234375,135.830671875,77.6124375],[0.25558857327929,-0.245486949695007,-0.647753398495225,0.674408017061174],[0,0,0,0],[8.999999E+09,8.999999E+09,8.999999E+09,8.999999E+09,8.999999E+09,8.999999E+09]];
	LOCAL CONST Robtarget Tr_meulage_bavure_P79 :=[[-40.65559765625,140.627546875,76.360421875],[0.255461049701821,-0.244928827106411,-0.64727981376299,0.675113593725138],[0,0,0,0],[8.999999E+09,8.999999E+09,8.999999E+09,8.999999E+09,8.999999E+09,8.999999E+09]];
	LOCAL CONST Robtarget Tr_meulage_bavure_P80 :=[[-42.83280859375,142.613078125,75.8436953125],[0.253983770206129,-0.242945633310523,-0.647128802853442,0.676530839093607],[0,0,0,0],[8.999999E+09,8.999999E+09,8.999999E+09,8.999999E+09,8.999999E+09,8.999999E+09]];
	LOCAL CONST Robtarget Tr_meulage_bavure_P81 :=[[-44.122875,143.761078125,75.5405390625],[0.249740750005927,-0.238196024814374,-0.647777432785459,0.679173474984843],[0,0,0,0],[8.999999E+09,8.999999E+09,8.999999E+09,8.999999E+09,8.999999E+09,8.999999E+09]];
	LOCAL CONST Robtarget Tr_meulage_bavure_P82 :=[[-44.80824609375,144.422234375,75.374046875],[0.24078412187225,-0.228863579953277,-0.649812221033629,0.683658208332586],[0,0,0,0],[8.999999E+09,8.999999E+09,8.999999E+09,8.999999E+09,8.999999E+09,8.999999E+09]];
	LOCAL CONST Robtarget Tr_meulage_bavure_P83 :=[[-48.56875390625,148.05365625,74.4601171875],[0.224736624931076,-0.212766667362191,-0.653751568256924,0.690530724642856],[0,0,0,0],[8.999999E+09,8.999999E+09,8.999999E+09,8.999999E+09,8.999999E+09,8.999999E+09]];
	LOCAL CONST Robtarget Tr_meulage_bavure_P84 :=[[-51.00261328125,150.07946875,73.9030390625],[0.19914887448737,-0.187706517706813,-0.659707701360471,0.699922665561332],[0,0,0,0],[8.999999E+09,8.999999E+09,8.999999E+09,8.999999E+09,8.999999E+09,8.999999E+09]];
	LOCAL CONST Robtarget Tr_meulage_bavure_P85 :=[[-51.525328125,150.455921875,73.789625],[0.162103514357927,-0.152050112590495,-0.667017208479469,0.711119720923476],[0,0,0,0],[8.999999E+09,8.999999E+09,8.999999E+09,8.999999E+09,8.999999E+09,8.999999E+09]];
	LOCAL CONST Robtarget Tr_meulage_bavure_P86 :=[[-52.99160546875,150.87928125,73.5386171875],[0.113314523462914,-0.105736494289701,-0.673992829034353,0.722297223418425],[0,0,0,0],[8.999999E+09,8.999999E+09,8.999999E+09,8.999999E+09,8.999999E+09,8.999999E+09]];
	LOCAL CONST Robtarget Tr_meulage_bavure_P87 :=[[-55.19370703125,151.642546875,73.148125],[0.0551646810886564,-0.0511960310796987,-0.678319780148977,0.730902250797408],[0,0,0,0],[8.999999E+09,8.999999E+09,8.999999E+09,8.999999E+09,8.999999E+09,8.999999E+09]];
	LOCAL CONST Robtarget Tr_meulage_bavure_P88 :=[[-56.68248828125,151.275078125,72.977890625],[0.00739546197339107,-0.00682503837738053,0.678163027934926,-0.734842590991758],[0,0,0,0],[8.999999E+09,8.999999E+09,8.999999E+09,8.999999E+09,8.999999E+09,8.999999E+09]];
	LOCAL CONST Robtarget Tr_meulage_bavure_P89 :=[[-58.1905,150.533015625,72.8447109375],[0.0688699449635165,-0.0631978054838895,0.673154071971728,-0.733571103200382],[0,0,0,0],[8.999999E+09,8.999999E+09,8.999999E+09,8.999999E+09,8.999999E+09,8.999999E+09]];
	LOCAL CONST Robtarget Tr_meulage_bavure_P90 :=[[-58.4362734375,150.44484375,72.81953125],[0.125454565902135,-0.114472434988728,0.664243148838317,-0.727968579502863],[0,0,0,0],[8.999999E+09,8.999999E+09,8.999999E+09,8.999999E+09,8.999999E+09,8.999999E+09]];
	LOCAL CONST Robtarget Tr_meulage_bavure_P91 :=[[-58.7546640625,150.150546875,72.806015625],[0.175518659022365,-0.159267010428992,0.65284354926812,-0.719459880676474],[0,0,0,0],[8.999999E+09,8.999999E+09,8.999999E+09,8.999999E+09,8.999999E+09,8.999999E+09]];
	LOCAL CONST Robtarget Tr_meulage_bavure_P92 :=[[-60.00348828125,148.9610625,72.7567578125],[0.218479538760072,-0.197189263800458,0.640336699469111,-0.709473041558328],[0,0,0,0],[8.999999E+09,8.999999E+09,8.999999E+09,8.999999E+09,8.999999E+09,8.999999E+09]];
	LOCAL CONST Robtarget Tr_meulage_bavure_P93 :=[[-61.4485,147.2434375,72.7359765625],[0.253948422262235,-0.228035670212907,0.628006378542772,-0.699369659372398],[0,0,0,0],[8.999999E+09,8.999999E+09,8.999999E+09,8.999999E+09,8.999999E+09,8.999999E+09]];
	LOCAL CONST Robtarget Tr_meulage_bavure_P94 :=[[-62.95536328125,145.01390625,72.7608359375],[0.281548074267506,-0.25161178289012,0.617024443898413,-0.690436838689078],[0,0,0,0],[8.999999E+09,8.999999E+09,8.999999E+09,8.999999E+09,8.999999E+09,8.999999E+09]];
	LOCAL CONST Robtarget Tr_meulage_bavure_P95 :=[[-64.22771484375,143.217890625,72.772640625],[0.301300782523362,-0.268077221042492,0.608261438776506,-0.683644983969369],[0,0,0,0],[8.999999E+09,8.999999E+09,8.999999E+09,8.999999E+09,8.999999E+09,8.999999E+09]];
	LOCAL CONST Robtarget Tr_meulage_bavure_P96 :=[[-64.75654296875,142.5368125,72.770609375],[0.313902551231965,-0.278168991851721,0.602069435683412,-0.679411211946137],[0,0,0,0],[8.999999E+09,8.999999E+09,8.999999E+09,8.999999E+09,8.999999E+09,8.999999E+09]];
	LOCAL CONST Robtarget Tr_meulage_bavure_P97 :=[[-66.1481484375,140.852078125,72.75384375],[0.320731782943178,-0.283200918474212,0.598240915781166,-0.677522080725613],[0,0,0,0],[8.999999E+09,8.999999E+09,8.999999E+09,8.999999E+09,8.999999E+09,8.999999E+09]];
	LOCAL CONST Robtarget Tr_meulage_bavure_P98 :=[[-74.1771953125,131.099640625,72.66053125],[0.323552254080279,-0.284795435416734,0.596188523547865,-0.67732174277457],[0,0,0,0],[8.999999E+09,8.999999E+09,8.999999E+09,8.999999E+09,8.999999E+09,8.999999E+09]];
	LOCAL CONST Robtarget Tr_meulage_bavure_P99 :=[[-76.206828125,128.7145,72.6284375],[0.324069609428897,-0.284481064074341,0.595223363730784,-0.678054982797666],[0,0,0,0],[8.999999E+09,8.999999E+09,8.999999E+09,8.999999E+09,8.999999E+09,8.999999E+09]];
	LOCAL CONST Robtarget Tr_meulage_bavure_P100 :=[[-80.3780625,123.7802578125,72.5659140625],[0.323587469228673,-0.283414490599376,0.594795959714879,-0.679106134991678],[0,0,0,0],[8.999999E+09,8.999999E+09,8.999999E+09,8.999999E+09,8.999999E+09,8.999999E+09]];
	LOCAL CONST Robtarget Tr_meulage_bavure_P101 :=[[-84.917109375,118.15028125,72.525546875],[0.322882334381622,-0.282277900571584,0.594577924449451,-0.680105342392307],[0,0,0,0],[8.999999E+09,8.999999E+09,8.999999E+09,8.999999E+09,8.999999E+09,8.999999E+09]];
	LOCAL CONST Robtarget Tr_meulage_bavure_P102 :=[[-85.1642109375,117.853390625,72.522328125],[0.322273215954625,-0.281343069248563,0.594430995277322,-0.680909570734377],[0,0,0,0],[8.999999E+09,8.999999E+09,8.999999E+09,8.999999E+09,8.999999E+09,8.999999E+09]];
	LOCAL CONST Robtarget Tr_meulage_bavure_P103 :=[[-94.3469140625,107.0483515625,72.3786015625],[0.321784084510284,-0.280625247640009,0.594342685922141,-0.681513936052461],[0,0,0,0],[8.999999E+09,8.999999E+09,8.999999E+09,8.999999E+09,8.999999E+09,8.999999E+09]];
	LOCAL CONST Robtarget Tr_meulage_bavure_P104 :=[[-96.91753125,103.8055625,72.3615],[0.321373274666824,-0.280079324681988,0.594323696994459,-0.681948776233555],[0,0,0,0],[8.999999E+09,8.999999E+09,8.999999E+09,8.999999E+09,8.999999E+09,8.999999E+09]];
	LOCAL CONST Robtarget Tr_meulage_bavure_P105 :=[[-97.6902265625,102.899234375,72.3491015625],[0.320985475815331,-0.279649176065806,0.594390211898772,-0.682249909227003],[0,0,0,0],[8.999999E+09,8.999999E+09,8.999999E+09,8.999999E+09,8.999999E+09,8.999999E+09]];
	LOCAL CONST Robtarget Tr_meulage_bavure_P106 :=[[-100.5085703125,99.583,72.304984375],[0.320585228347759,-0.279297429699102,0.594551080212047,-0.682441990316671],[0,0,0,0],[8.999999E+09,8.999999E+09,8.999999E+09,8.999999E+09,8.999999E+09,8.999999E+09]];
	LOCAL CONST Robtarget Tr_meulage_bavure_P107 :=[[-105.7713671875,93.279921875,72.2343359375],[0.320150595649433,-0.278997572954701,0.594808363925635,-0.682544475177119],[0,0,0,0],[8.999999E+09,8.999999E+09,8.999999E+09,8.999999E+09,8.999999E+09,8.999999E+09]];
	LOCAL CONST Robtarget Tr_meulage_bavure_P108 :=[[-108.448953125,90.1716484375,72.1879296875],[0.319667753250009,-0.278733358327595,0.59516388008965,-0.68256882314104],[0,0,0,0],[8.999999E+09,8.999999E+09,8.999999E+09,8.999999E+09,8.999999E+09,8.999999E+09]];
	LOCAL CONST Robtarget Tr_meulage_bavure_P109 :=[[-110.28228125,88.0006171875,72.160703125],[0.319136566210563,-0.278496654835877,0.595609932286619,-0.682524925489235],[0,0,0,0],[8.999999E+09,8.999999E+09,8.999999E+09,8.999999E+09,8.999999E+09,8.999999E+09]];
	LOCAL CONST Robtarget Tr_meulage_bavure_P110 :=[[-111.2027890625,86.8564375,72.1527734375],[0.318563922768677,-0.278291926129409,0.596142453233964,-0.682411024539907],[0,0,0,0],[8.999999E+09,8.999999E+09,8.999999E+09,8.999999E+09,8.999999E+09,8.999999E+09]];
	LOCAL CONST Robtarget Tr_meulage_bavure_P111 :=[[-121.120125,74.994265625,72.018],[0.317972009866905,-0.278135222761113,0.596749280210868,-0.682220562112164],[0,0,0,0],[8.999999E+09,8.999999E+09,8.999999E+09,8.999999E+09,8.999999E+09,8.999999E+09]];
	LOCAL CONST Robtarget Tr_meulage_bavure_P112 :=[[-121.641921875,74.3759609375,72.0102890625],[0.317384461486392,-0.278041917112747,0.597415547098783,-0.681949015704197],[0,0,0,0],[8.999999E+09,8.999999E+09,8.999999E+09,8.999999E+09,8.999999E+09,8.999999E+09]];
	LOCAL CONST Robtarget Tr_meulage_bavure_P113 :=[[-121.727546875,74.276140625,72.0088515625],[0.316815542110126,-0.278024861433691,0.598135777897993,-0.681589084346724],[0,0,0,0],[8.999999E+09,8.999999E+09,8.999999E+09,8.999999E+09,8.999999E+09,8.999999E+09]];
	LOCAL CONST Robtarget Tr_meulage_bavure_P114 :=[[-121.7964765625,74.1953125,72.0077421875],[0.316280561105061,-0.278095375211244,0.5989013799309,-0.681136334422155],[0,0,0,0],[8.999999E+09,8.999999E+09,8.999999E+09,8.999999E+09,8.999999E+09,8.999999E+09]];
	LOCAL CONST Robtarget Tr_meulage_bavure_P115 :=[[-122.4996015625,73.3805859375,71.9953984375],[0.315778556845359,-0.278253275545646,0.59971301993204,-0.680590413838436],[0,0,0,0],[8.999999E+09,8.999999E+09,8.999999E+09,8.999999E+09,8.999999E+09,8.999999E+09]];
	LOCAL CONST Robtarget Tr_meulage_bavure_P116 :=[[-127.177609375,67.9651953125,71.91271875],[0.315290892330133,-0.278480900164475,0.600576579825214,-0.679961626286881],[0,0,0,0],[8.999999E+09,8.999999E+09,8.999999E+09,8.999999E+09,8.999999E+09,8.999999E+09]];
	LOCAL CONST Robtarget Tr_meulage_bavure_P117 :=[[-127.844921875,67.216296875,71.898421875],[0.314778701374699,-0.278739951044396,0.601503608348698,-0.679273006968569],[0,0,0,0],[8.999999E+09,8.999999E+09,8.999999E+09,8.999999E+09,8.999999E+09,8.999999E+09]];
	LOCAL CONST Robtarget Tr_meulage_bavure_P118 :=[[-129.4959765625,65.23797265625,71.8763515625],[0.314199815612523,-0.278992829919956,0.602511121151723,-0.678543901019532],[0,0,0,0],[8.999999E+09,8.999999E+09,8.999999E+09,8.999999E+09,8.999999E+09,8.999999E+09]];
	LOCAL CONST Robtarget Tr_meulage_bavure_P119 :=[[-132.03303125,62.2335546875,71.838671875],[0.313578720275502,-0.279253983738639,0.603581917538199,-0.677771692812107],[0,0,0,0],[8.999999E+09,8.999999E+09,8.999999E+09,8.999999E+09,8.999999E+09,8.999999E+09]];
	LOCAL CONST Robtarget Tr_meulage_bavure_P120 :=[[-134.127640625,59.69999609375,71.813203125],[0.313042074049291,-0.279627654723897,0.604654879707455,-0.676908790779448],[0,0,0,0],[8.999999E+09,8.999999E+09,8.999999E+09,8.999999E+09,8.999999E+09,8.999999E+09]];
	LOCAL CONST Robtarget Tr_meulage_bavure_P121 :=[[-140.83225,52.17749609375,71.66934375],[0.312853762381832,-0.280344883483948,0.605613869255388,-0.67584103976706],[0,0,0,0],[8.999999E+09,8.999999E+09,8.999999E+09,8.999999E+09,8.999999E+09,8.999999E+09]];
	LOCAL CONST Robtarget Tr_meulage_bavure_P122 :=[[-141.791875,51.09122265625,71.6497734375],[0.313381105843567,-0.281725991447276,0.606290562297042,-0.674414191956879],[0,0,0,0],[8.999999E+09,8.999999E+09,8.999999E+09,8.999999E+09,8.999999E+09,8.999999E+09]];
	LOCAL CONST Robtarget Tr_meulage_bavure_P123 :=[[-142.175171875,50.64507421875,71.6432578125],[0.31501556371639,-0.284110651956207,0.606493792710147,-0.67246681067955],[0,0,0,0],[8.999999E+09,8.999999E+09,8.999999E+09,8.999999E+09,8.999999E+09,8.999999E+09]];
	LOCAL CONST Robtarget Tr_meulage_bavure_P124 :=[[-142.260234375,50.5402109375,71.6424296875],[0.318050077820343,-0.287756674470804,0.606065806488869,-0.669869003985835],[0,0,0,0],[8.999999E+09,8.999999E+09,8.999999E+09,8.999999E+09,8.999999E+09,8.999999E+09]];
	LOCAL CONST Robtarget Tr_meulage_bavure_P125 :=[[-149.162828125,42.43656640625,71.5324375],[0.322613935718291,-0.29276739930339,0.6048968443299,-0.666563804976848],[0,0,0,0],[8.999999E+09,8.999999E+09,8.999999E+09,8.999999E+09,8.999999E+09,8.999999E+09]];
	LOCAL CONST Robtarget Tr_meulage_bavure_P126 :=[[-150.8765,40.4939296875,71.49778125],[0.328865189677666,-0.29926998454819,0.602848120897509,-0.662464569993854],[0,0,0,0],[8.999999E+09,8.999999E+09,8.999999E+09,8.999999E+09,8.999999E+09,8.999999E+09]];
	LOCAL CONST Robtarget Tr_meulage_bavure_P127 :=[[-155.496890625,35.53946875,71.37428125],[0.337148295607245,-0.307555587024709,0.599670598353181,-0.657370337884023],[0,0,0,0],[8.999999E+09,8.999999E+09,8.999999E+09,8.999999E+09,8.999999E+09,8.999999E+09]];
	LOCAL CONST Robtarget Tr_meulage_bavure_P128 :=[[-156.39446875,34.56391796875,71.351671875],[0.348390803658434,-0.318439565768407,0.594786388170789,-0.650729777500773],[0,0,0,0],[8.999999E+09,8.999999E+09,8.999999E+09,8.999999E+09,8.999999E+09,8.999999E+09]];
	LOCAL CONST Robtarget Tr_meulage_bavure_P129 :=[[-156.51775,34.41030859375,71.3506484375],[0.364395126457295,-0.33353440521878,0.587046466427617,-0.641363733465165],[0,0,0,0],[8.999999E+09,8.999999E+09,8.999999E+09,8.999999E+09,8.999999E+09,8.999999E+09]];
	LOCAL CONST Robtarget Tr_meulage_bavure_P130 :=[[-157.774984375,32.659912109375,71.3597421875],[0.387792497602994,-0.355202422143889,0.574501826401859,-0.627212778542397],[0,0,0,0],[8.999999E+09,8.999999E+09,8.999999E+09,8.999999E+09,8.999999E+09,8.999999E+09]];
	LOCAL CONST Robtarget Tr_meulage_bavure_P131 :=[[-157.900296875,32.39592578125,71.3701484375],[0.421582073394979,-0.386117593908087,0.55415673640107,-0.605055427682403],[0,0,0,0],[8.999999E+09,8.999999E+09,8.999999E+09,8.999999E+09,8.999999E+09,8.999999E+09]];
	LOCAL CONST Robtarget Tr_meulage_bavure_P132 :=[[-159.11453125,29.7500703125,71.4803203125],[0.467558162831586,-0.427798010222454,0.522177346335793,-0.570709248035258],[0,0,0,0],[8.999999E+09,8.999999E+09,8.999999E+09,8.999999E+09,8.999999E+09,8.999999E+09]];
	LOCAL CONST Robtarget Tr_meulage_bavure_P133 :=[[-159.110828125,29.73805078125,71.4821171875],[0.523327030125884,-0.477872362269479,0.475742762115945,-0.520994864862314],[0,0,0,0],[8.999999E+09,8.999999E+09,8.999999E+09,8.999999E+09,8.999999E+09,8.999999E+09]];
	LOCAL CONST Robtarget Tr_meulage_bavure_P134 :=[[-158.46065625,25.9234296875,71.9783671875],[0.580045010263931,-0.528050136917584,0.417544472176329,-0.458658318058474],[0,0,0,0],[8.999999E+09,8.999999E+09,8.999999E+09,8.999999E+09,8.999999E+09,8.999999E+09]];
	LOCAL CONST Robtarget Tr_meulage_bavure_P135 :=[[-157.70496875,24.849541015625,72.1985546875],[0.626913573831798,-0.568350297054104,0.357909446496227,-0.394788726906834],[0,0,0,0],[8.999999E+09,8.999999E+09,8.999999E+09,8.999999E+09,8.999999E+09,8.999999E+09]];
	LOCAL CONST Robtarget Tr_meulage_bavure_P136 :=[[-156.218546875,23.191529296875,72.5834296875],[0.659328155046374,-0.594594057421879,0.308171772780454,-0.341722766732163],[0,0,0,0],[8.999999E+09,8.999999E+09,8.999999E+09,8.999999E+09,8.999999E+09,8.999999E+09]];
	LOCAL CONST Robtarget Tr_meulage_bavure_P137 :=[[-153.62478125,21.171771484375,73.1623359375],[0.679265187433453,-0.608685069063752,0.27361691958939,-0.30534418801455],[0,0,0,0],[8.999999E+09,8.999999E+09,8.999999E+09,8.999999E+09,8.999999E+09,8.999999E+09]];
	LOCAL CONST Robtarget Tr_meulage_bavure_P138 :=[[-153.484375,21.060689453125,73.193859375],[0.690384664982347,-0.61409260905778,0.254174858961978,-0.285752380444118],[0,0,0,0],[8.999999E+09,8.999999E+09,8.999999E+09,8.999999E+09,8.999999E+09,8.999999E+09]];
	LOCAL CONST Robtarget Tr_meulage_bavure_P139 :=[[-153.401296875,21.000048828125,73.21196875],[0.695409570999413,-0.613428349879028,0.247616227090714,-0.280708731977588],[0,0,0,0],[8.999999E+09,8.999999E+09,8.999999E+09,8.999999E+09,8.999999E+09,8.999999E+09]];
	LOCAL CONST Robtarget Tr_meulage_bavure_P140 :=[[-148.92934375,17.9339609375,74.1658828125],[0.695839173381053,-0.608223531793992,0.251355083683277,-0.287563214036476],[0,0,0,0],[8.999999E+09,8.999999E+09,8.999999E+09,8.999999E+09,8.999999E+09,8.999999E+09]];
	LOCAL CONST Robtarget Tr_meulage_bavure_P141 :=[[-146.0503125,15.580923828125,74.82025],[0.692424286864386,-0.599357265004037,0.262863869143026,-0.303680855745608],[0,0,0,0],[8.999999E+09,8.999999E+09,8.999999E+09,8.999999E+09,8.999999E+09,8.999999E+09]];
	LOCAL CONST Robtarget Tr_meulage_bavure_P142 :=[[-142.48975,12.6240068359375,75.6345],[0.685619806404656,-0.587453392019438,0.279722174831166,-0.326465156147208],[0,0,0,0],[8.999999E+09,8.999999E+09,8.999999E+09,8.999999E+09,8.999999E+09,8.999999E+09]];
	LOCAL CONST Robtarget Tr_meulage_bavure_P143 :=[[-139.376109375,9.5127861328125,76.4023046875],[0.675861065996386,-0.573117464315947,0.299711859165122,-0.353441640220946],[0,0,0,0],[8.999999E+09,8.999999E+09,8.999999E+09,8.999999E+09,8.999999E+09,8.999999E+09]];
	LOCAL CONST Robtarget Tr_meulage_bavure_P144 :=[[-137.58640625,7.33159423828125,76.8853359375],[0.66368128168553,-0.55701826218761,0.320958153105769,-0.382418195023042],[0,0,0,0],[8.999999E+09,8.999999E+09,8.999999E+09,8.999999E+09,8.999999E+09,8.999999E+09]];
	LOCAL CONST Robtarget Tr_meulage_bavure_P145 :=[[-137.177515625,6.68771044921875,77.011140625],[0.649458964561094,-0.539670774564678,0.342358450394871,-0.412006310479845],[0,0,0,0],[8.999999E+09,8.999999E+09,8.999999E+09,8.999999E+09,8.999999E+09,8.999999E+09]];
	LOCAL CONST Robtarget Tr_meulage_bavure_P146 :=[[-136.13084375,4.8995556640625,77.34803125],[0.633192679276466,-0.521244216590471,0.363642009198451,-0.441741991130332],[0,0,0,0],[8.999999E+09,8.999999E+09,8.999999E+09,8.999999E+09,8.999999E+09,8.999999E+09]];
	LOCAL CONST Robtarget Tr_meulage_bavure_P147 :=[[-135.970046875,4.36547998046875,77.4273203125],[0.61445370048275,-0.501528048585026,0.38510480597616,-0.471816229966302],[0,0,0,0],[8.999999E+09,8.999999E+09,8.999999E+09,8.999999E+09,8.999999E+09,8.999999E+09]];
	LOCAL CONST Robtarget Tr_meulage_bavure_P148 :=[[-135.78753125,3.64960522460937,77.5289453125],[0.592743447722771,-0.480234265639163,0.407011610910351,-0.502366204946051],[0,0,0,0],[8.999999E+09,8.999999E+09,8.999999E+09,8.999999E+09,8.999999E+09,8.999999E+09]];
	LOCAL CONST Robtarget Tr_meulage_bavure_P149 :=[[-134.88234375,1.00417333984375,77.9369453125],[0.568318790839792,-0.457637960071897,0.428868267754265,-0.532591079903792],[0,0,0,0],[8.999999E+09,8.999999E+09,8.999999E+09,8.999999E+09,8.999999E+09,8.999999E+09]];
	LOCAL CONST Robtarget Tr_meulage_bavure_P150 :=[[-134.92671875,-2.50852124023438,78.30353125],[0.542919642858546,-0.435166547003873,0.449203566140403,-0.560432416919131],[0,0,0,0],[8.999999E+09,8.999999E+09,8.999999E+09,8.999999E+09,8.999999E+09,8.999999E+09]];
	LOCAL CONST Robtarget Tr_meulage_bavure_P151 :=[[-135.0774375,-3.41068676757813,78.3781015625],[0.51995176016308,-0.415511311571464,0.465917518997469,-0.583027771680491],[0,0,0,0],[8.999999E+09,8.999999E+09,8.999999E+09,8.999999E+09,8.999999E+09,8.999999E+09]];
	LOCAL CONST Robtarget Tr_meulage_bavure_P152 :=[[-135.7479375,-4.8949423828125,78.44140625],[0.503539186635306,-0.401869770635279,0.477082609198778,-0.597780192857115],[0,0,0,0],[8.999999E+09,8.999999E+09,8.999999E+09,8.999999E+09,8.999999E+09,8.999999E+09]];
	LOCAL CONST Robtarget Tr_meulage_bavure_P153 :=[[-136.1586875,-6.201587890625,78.5223671875],[0.497122928447713,-0.396917530602435,0.481420295220917,-0.602959175451739],[0,0,0,0],[8.999999E+09,8.999999E+09,8.999999E+09,8.999999E+09,8.999999E+09,8.999999E+09]];
	LOCAL CONST Robtarget Tr_meulage_bavure_P154 :=[[-137.350390625,-8.31646484375,78.5793515625],[0.502558839704465,-0.402120826785359,0.478152740428553,-0.597581300009485],[0,0,0,0],[8.999999E+09,8.999999E+09,8.999999E+09,8.999999E+09,8.999999E+09,8.999999E+09]];
	LOCAL CONST Robtarget Tr_meulage_bavure_P155 :=[[-141.369546875,-14.628466796875,78.6844296875],[0.51977323559267,-0.417475366036216,0.466746494477794,-0.581117726633034],[0,0,0,0],[8.999999E+09,8.999999E+09,8.999999E+09,8.999999E+09,8.999999E+09,8.999999E+09]];
	LOCAL CONST Robtarget Tr_meulage_bavure_P156 :=[[-141.391140625,-14.6641904296875,78.6851875],[0.546680183368139,-0.441425164956329,0.447008838598085,-0.553595248418054],[0,0,0,0],[8.999999E+09,8.999999E+09,8.999999E+09,8.999999E+09,8.999999E+09,8.999999E+09]];
	LOCAL CONST Robtarget Tr_meulage_bavure_P157 :=[[-141.5636875,-15.4239521484375,78.741578125],[0.57937844774719,-0.470962969064101,0.419598302129201,-0.516189655946993],[0,0,0,0],[8.999999E+09,8.999999E+09,8.999999E+09,8.999999E+09,8.999999E+09,8.999999E+09]];
	LOCAL CONST Robtarget Tr_meulage_bavure_P158 :=[[-141.870421875,-17.969013671875,78.96859375],[0.612949481335847,-0.502185140696095,0.386590570116858,-0.471858823050796],[0,0,0,0],[8.999999E+09,8.999999E+09,8.999999E+09,8.999999E+09,8.999999E+09,8.999999E+09]];
	LOCAL CONST Robtarget Tr_meulage_bavure_P159 :=[[-140.856453125,-20.692720703125,79.4001875],[0.642898315529926,-0.531378077680427,0.351449713119889,-0.425208411955109],[0,0,0,0],[8.999999E+09,8.999999E+09,8.999999E+09,8.999999E+09,8.999999E+09,8.999999E+09]];
	LOCAL CONST Robtarget Tr_meulage_bavure_P160 :=[[-140.265578125,-21.746759765625,79.5951015625],[0.666527894006695,-0.55617016277201,0.318035430054266,-0.381141419663823],[0,0,0,0],[8.999999E+09,8.999999E+09,8.999999E+09,8.999999E+09,8.999999E+09,8.999999E+09]];
	LOCAL CONST Robtarget Tr_meulage_bavure_P161 :=[[-139.10271875,-23.3570625,79.9294375],[0.683199867898617,-0.575814775689324,0.28941388073797,-0.343387376351192],[0,0,0,0],[8.999999E+09,8.999999E+09,8.999999E+09,8.999999E+09,8.999999E+09,8.999999E+09]];
	LOCAL CONST Robtarget Tr_meulage_bavure_P162 :=[[-138.114796875,-24.308181640625,80.169234375],[0.693705019907949,-0.590697097940034,0.267189731665087,-0.313783255022432],[0,0,0,0],[8.999999E+09,8.999999E+09,8.999999E+09,8.999999E+09,8.999999E+09,8.999999E+09]];
	LOCAL CONST Robtarget Tr_meulage_bavure_P163 :=[[-137.169578125,-25.168494140625,80.3933828125],[0.699360303058629,-0.601660810401763,0.2516563023373,-0.292521009888785],[0,0,0,0],[8.999999E+09,8.999999E+09,8.999999E+09,8.999999E+09,8.999999E+09,8.999999E+09]];
	LOCAL CONST Robtarget Tr_meulage_bavure_P164 :=[[-133.03959375,-28.32869921875,81.309234375],[0.701502624120611,-0.60963669392408,0.242114974028717,-0.27859919081772],[0,0,0,0],[8.999999E+09,8.999999E+09,8.999999E+09,8.999999E+09,8.999999E+09,8.999999E+09]];
	LOCAL CONST Robtarget Tr_meulage_bavure_P165 :=[[-131.817,-29.272169921875,81.5811953125],[0.701308692921814,-0.615462063748357,0.237249993690512,-0.270342386267419],[0,0,0,0],[8.999999E+09,8.999999E+09,8.999999E+09,8.999999E+09,8.999999E+09,8.999999E+09]];
	LOCAL CONST Robtarget Tr_meulage_bavure_P166 :=[[-130.923859375,-30.038609375,81.7880625],[0.699746882491147,-0.619847322229403,0.235503463991653,-0.265860331785116],[0,0,0,0],[8.999999E+09,8.999999E+09,8.999999E+09,8.999999E+09,8.999999E+09,8.999999E+09]];
	LOCAL CONST Robtarget Tr_meulage_bavure_P167 :=[[-129.1705546875,-31.674556640625,82.208109375],[0.697585551602146,-0.623362970756538,0.235386055708575,-0.263413002077486],[0,0,0,0],[8.999999E+09,8.999999E+09,8.999999E+09,8.999999E+09,8.999999E+09,8.999999E+09]];
	LOCAL CONST Robtarget Tr_meulage_bavure_P168 :=[[-127.9752109375,-32.7016171875,82.4851171875],[0.695351286512787,-0.626438529408559,0.235754440933495,-0.261689130071521],[0,0,0,0],[8.999999E+09,8.999999E+09,8.999999E+09,8.999999E+09,8.999999E+09,8.999999E+09]];
	LOCAL CONST Robtarget Tr_meulage_bavure_P169 :=[[-124.597125,-35.74508984375,83.2828984375],[0.693366797217647,-0.629341164182628,0.235876839488228,-0.259873623468103],[0,0,0,0],[8.999999E+09,8.999999E+09,8.999999E+09,8.999999E+09,8.999999E+09,8.999999E+09]];
	LOCAL CONST Robtarget Tr_meulage_bavure_P170 :=[[-122.34146875,-37.836171875,83.8218515625],[0.691746366234012,-0.632154336056749,0.23549830069305,-0.257698293702882],[0,0,0,0],[8.999999E+09,8.999999E+09,8.999999E+09,8.999999E+09,8.999999E+09,8.999999E+09]];
	LOCAL CONST Robtarget Tr_meulage_bavure_P171 :=[[-121.9502578125,-38.14978515625,83.9101171875],[0.690450060150475,-0.634857419927956,0.234697164664331,-0.255248921053836],[0,0,0,0],[8.999999E+09,8.999999E+09,8.999999E+09,8.999999E+09,8.999999E+09,8.999999E+09]];
	LOCAL CONST Robtarget Tr_meulage_bavure_P172 :=[[-121.340203125,-38.63997265625,84.0478828125],[0.68935992214546,-0.637373038283842,0.233733920717123,-0.252798263670128],[0,0,0,0],[8.999999E+09,8.999999E+09,8.999999E+09,8.999999E+09,8.999999E+09,8.999999E+09]];
	LOCAL CONST Robtarget Tr_meulage_bavure_P173 :=[[-114.677,-44.1038203125,85.56425],[0.688331388926613,-0.639589566154633,0.232957524680154,-0.250710744842307],[0,0,0,0],[8.999999E+09,8.999999E+09,8.999999E+09,8.999999E+09,8.999999E+09,8.999999E+09]];
	LOCAL CONST Robtarget Tr_meulage_bavure_P174 :=[[-114.170234375,-44.43026953125,85.670125],[0.687254698142657,-0.641428457268899,0.232638226117913,-0.249258841037176],[0,0,0,0],[8.999999E+09,8.999999E+09,8.999999E+09,8.999999E+09,8.999999E+09,8.999999E+09]];
	LOCAL CONST Robtarget Tr_meulage_bavure_P175 :=[[-113.8066171875,-44.81165234375,85.761703125],[0.686078928414305,-0.6428718985253,0.232890352942438,-0.24854277213128],[0,0,0,0],[8.999999E+09,8.999999E+09,8.999999E+09,8.999999E+09,8.999999E+09,8.999999E+09]];
	LOCAL CONST Robtarget Tr_meulage_bavure_P176 :=[[-112.3647265625,-46.11738671875,86.1029375],[0.684818543953459,-0.643963957147717,0.233652689256344,-0.248476164964362],[0,0,0,0],[8.999999E+09,8.999999E+09,8.999999E+09,8.999999E+09,8.999999E+09,8.999999E+09]];
	LOCAL CONST Robtarget Tr_meulage_bavure_P177 :=[[-109.447421875,-48.8080703125,86.798515625],[0.683537513098722,-0.644783386675879,0.234742247755828,-0.248851219752163],[0,0,0,0],[8.999999E+09,8.999999E+09,8.999999E+09,8.999999E+09,8.999999E+09,8.999999E+09]];
	LOCAL CONST Robtarget Tr_meulage_bavure_P178 :=[[-108.7766484375,-49.5145859375,86.9677734375],[0.682306788344517,-0.645415725116894,0.235954985338503,-0.249441843411908],[0,0,0,0],[8.999999E+09,8.999999E+09,8.999999E+09,8.999999E+09,8.999999E+09,8.999999E+09]];
	LOCAL CONST Robtarget Tr_meulage_bavure_P179 :=[[-102.3894296875,-55.16411328125,88.4650703125],[0.68117096001414,-0.645914559160078,0.23716308907001,-0.250108325893457],[0,0,0,0],[8.999999E+09,8.999999E+09,8.999999E+09,8.999999E+09,8.999999E+09,8.999999E+09]];
	LOCAL CONST Robtarget Tr_meulage_bavure_P180 :=[[-102.30465625,-55.238484375,88.484875],[0.680134384325639,-0.64629646824612,0.238342117209733,-0.250820911318332],[0,0,0,0],[8.999999E+09,8.999999E+09,8.999999E+09,8.999999E+09,8.999999E+09,8.999999E+09]];
	LOCAL CONST Robtarget Tr_meulage_bavure_P181 :=[[-102.223609375,-55.3030546875,88.5031171875],[0.679183503282743,-0.64655001407483,0.239525705944634,-0.25161535000898],[0,0,0,0],[8.999999E+09,8.999999E+09,8.999999E+09,8.999999E+09,8.999999E+09,8.999999E+09]];
	LOCAL CONST Robtarget Tr_meulage_bavure_P182 :=[[-99.80740625,-57.17198828125,89.0410546875],[0.678306891584764,-0.646668902525575,0.240737976791992,-0.252515975465084],[0,0,0,0],[8.999999E+09,8.999999E+09,8.999999E+09,8.999999E+09,8.999999E+09,8.999999E+09]];
	LOCAL CONST Robtarget Tr_meulage_bavure_P183 :=[[-97.863984375,-58.84211328125,89.4914453125],[0.677515026654867,-0.646669197445363,0.241944971540456,-0.253485637617822],[0,0,0,0],[8.999999E+09,8.999999E+09,8.999999E+09,8.999999E+09,8.999999E+09,8.999999E+09]];
	LOCAL CONST Robtarget Tr_meulage_bavure_P184 :=[[-95.8647421875,-60.80031640625,89.980265625],[0.676834750837083,-0.646586947171256,0.24306685673286,-0.254437699575095],[0,0,0,0],[8.999999E+09,8.999999E+09,8.999999E+09,8.999999E+09,8.999999E+09,8.999999E+09]];
	LOCAL CONST Robtarget Tr_meulage_bavure_P185 :=[[-93.257390625,-63.2205234375,90.603578125],[0.676311199599883,-0.646456247730513,0.243999472969827,-0.255267973424791],[0,0,0,0],[8.999999E+09,8.999999E+09,8.999999E+09,8.999999E+09,8.999999E+09,8.999999E+09]];
	LOCAL CONST Robtarget Tr_meulage_bavure_P186 :=[[-90.280125,-66.1861796875,91.336765625],[0.675973858514008,-0.646328318796993,0.24464530849914,-0.255866605785312],[0,0,0,0],[8.999999E+09,8.999999E+09,8.999999E+09,8.999999E+09,8.999999E+09,8.999999E+09]];
	LOCAL CONST Robtarget Tr_meulage_bavure_P187 :=[[-88.7913046875,-67.3695234375,91.6716015625],[0.675853632208687,-0.646253783439602,0.244905858485635,-0.256123087010403],[0,0,0,0],[8.999999E+09,8.999999E+09,8.999999E+09,8.999999E+09,8.999999E+09,8.999999E+09]];
	LOCAL CONST Robtarget Tr_meulage_bavure_P188 :=[[-87.07525,-68.8335546875,92.068171875],[0.675996386951698,-0.646297396802448,0.244644219104513,-0.255886235998288],[0,0,0,0],[8.999999E+09,8.999999E+09,8.999999E+09,8.999999E+09,8.999999E+09,8.999999E+09]];
	LOCAL CONST Robtarget Tr_meulage_bavure_P189 :=[[-86.91775,-68.9480546875,92.1024609375],[0.676464990856974,-0.646537623239098,0.243679868631024,-0.254959486007443],[0,0,0,0],[8.999999E+09,8.999999E+09,8.999999E+09,8.999999E+09,8.999999E+09,8.999999E+09]];
	LOCAL CONST Robtarget Tr_meulage_bavure_P190 :=[[-86.848328125,-69.0137421875,92.1191875],[0.677299843470152,-0.647047252818023,0.241864355419417,-0.253172684611724],[0,0,0,0],[8.999999E+09,8.999999E+09,8.999999E+09,8.999999E+09,8.999999E+09,8.999999E+09]];
	LOCAL CONST Robtarget Tr_meulage_bavure_P191 :=[[-86.3394375,-69.5110546875,92.2434921875],[0.678490801475779,-0.647854914545416,0.239161788877326,-0.250471317226355],[0,0,0,0],[8.999999E+09,8.999999E+09,8.999999E+09,8.999999E+09,8.999999E+09,8.999999E+09]];
	LOCAL CONST Robtarget Tr_meulage_bavure_P192 :=[[-83.4334375,-72.2495390625,92.9425546875],[0.67994869521465,-0.648902111696461,0.235744167009118,-0.247023296538901],[0,0,0,0],[8.999999E+09,8.999999E+09,8.999999E+09,8.999999E+09,8.999999E+09,8.999999E+09]];
	LOCAL CONST Robtarget Tr_meulage_bavure_P193 :=[[-83.196703125,-72.4797109375,93.0002578125],[0.681484103007736,-0.650055693742827,0.232029481784419,-0.243247470620204],[0,0,0,0],[8.999999E+09,8.999999E+09,8.999999E+09,8.999999E+09,8.999999E+09,8.999999E+09]];
	LOCAL CONST Robtarget Tr_meulage_bavure_P194 :=[[-79.8956484375,-75.0584140625,93.7378828125],[0.682867266907574,-0.651132432749633,0.228584282130694,-0.239725002389239],[0,0,0,0],[8.999999E+09,8.999999E+09,8.999999E+09,8.999999E+09,8.999999E+09,8.999999E+09]];
	LOCAL CONST Robtarget Tr_meulage_bavure_P195 :=[[-79.234328125,-75.5704609375,93.885171875],[0.68388915067614,-0.65196130464372,0.225963136394031,-0.23702900207717],[0,0,0,0],[8.999999E+09,8.999999E+09,8.999999E+09,8.999999E+09,8.999999E+09,8.999999E+09]];
	LOCAL CONST Robtarget Tr_meulage_bavure_P196 :=[[-78.9871015625,-75.752703125,93.939265625],[0.684415027540741,-0.652445177099004,0.224532465200286,-0.235534568647023],[0,0,0,0],[8.999999E+09,8.999999E+09,8.999999E+09,8.999999E+09,8.999999E+09,8.999999E+09]];
	LOCAL CONST Robtarget Tr_meulage_bavure_P197 :=[[-76.2423203125,-77.6906640625,94.5307109375],[0.684413079535223,-0.652592681799339,0.224358014587739,-0.235297704011977],[0,0,0,0],[8.999999E+09,8.999999E+09,8.999999E+09,8.999999E+09,8.999999E+09,8.999999E+09]];
	LOCAL CONST Robtarget Tr_meulage_bavure_P198 :=[[-71.7864296875,-81.5057109375,95.561859375],[0.683949193545817,-0.65248998011423,0.225233844560194,-0.236093290381562],[0,0,0,0],[8.999999E+09,8.999999E+09,8.999999E+09,8.999999E+09,8.999999E+09,8.999999E+09]];
	LOCAL CONST Robtarget Tr_meulage_bavure_P199 :=[[-71.28534375,-81.9084921875,95.67503125],[0.683145646105371,-0.652257765804186,0.226808675474322,-0.237549274646313],[0,0,0,0],[8.999999E+09,8.999999E+09,8.999999E+09,8.999999E+09,8.999999E+09,8.999999E+09]];
	LOCAL CONST Robtarget Tr_meulage_bavure_P200 :=[[-70.9811015625,-82.1761484375,95.746203125],[0.682117506282282,-0.652012674447863,0.228748373119855,-0.239310179009598],[0,0,0,0],[8.999999E+09,8.999999E+09,8.999999E+09,8.999999E+09,8.999999E+09,8.999999E+09]];
	LOCAL CONST Robtarget Tr_meulage_bavure_P201 :=[[-70.84003125,-82.3231640625,95.7816328125],[0.6809365491792,-0.651846381667454,0.230824722028213,-0.241125814461182],[0,0,0,0],[8.999999E+09,8.999999E+09,8.999999E+09,8.999999E+09,8.999999E+09,8.999999E+09]];
	LOCAL CONST Robtarget Tr_meulage_bavure_P202 :=[[-68.6264375,-84.0588203125,96.2769453125],[0.679670182119976,-0.651795586230091,0.232887129263884,-0.24284674659381],[0,0,0,0],[8.999999E+09,8.999999E+09,8.999999E+09,8.999999E+09,8.999999E+09,8.999999E+09]];
	LOCAL CONST Robtarget Tr_meulage_bavure_P203 :=[[-65.645140625,-86.405171875,96.9449765625],[0.678371475041033,-0.651885163977952,0.234825351165252,-0.24436638329813],[0,0,0,0],[8.999999E+09,8.999999E+09,8.999999E+09,8.999999E+09,8.999999E+09,8.999999E+09]];
	LOCAL CONST Robtarget Tr_meulage_bavure_P204 :=[[-64.28871484375,-87.615203125,97.2640390625],[0.677085088697026,-0.652158930879137,0.236523127257573,-0.245563274556722],[0,0,0,0],[8.999999E+09,8.999999E+09,8.999999E+09,8.999999E+09,8.999999E+09,8.999999E+09]];
	LOCAL CONST Robtarget Tr_meulage_bavure_P205 :=[[-60.54962109375,-91.05371875,98.154484375],[0.675864267143362,-0.652626232752705,0.237891344165589,-0.246361931095021],[0,0,0,0],[8.999999E+09,8.999999E+09,8.999999E+09,8.999999E+09,8.999999E+09,8.999999E+09]];
	LOCAL CONST Robtarget Tr_meulage_bavure_P206 :=[[-58.79899609375,-92.5512265625,98.5594609375],[0.674719392306472,-0.653271954563657,0.238934469114216,-0.246778877733231],[0,0,0,0],[8.999999E+09,8.999999E+09,8.999999E+09,8.999999E+09,8.999999E+09,8.999999E+09]];
	LOCAL CONST Robtarget Tr_meulage_bavure_P207 :=[[-53.59029296875,-97.0586796875,99.76990625],[0.673638452552481,-0.654026138217555,0.239751941303447,-0.246941394691452],[0,0,0,0],[8.999999E+09,8.999999E+09,8.999999E+09,8.999999E+09,8.999999E+09,8.999999E+09]];
	LOCAL CONST Robtarget Tr_meulage_bavure_P208 :=[[-50.4647890625,-99.7672578125,100.4966484375],[0.672576465552345,-0.654814277335867,0.240498185100804,-0.247021827265207],[0,0,0,0],[8.999999E+09,8.999999E+09,8.999999E+09,8.999999E+09,8.999999E+09,8.999999E+09]];
	LOCAL CONST Robtarget Tr_meulage_bavure_P209 :=[[-49.2312265625,-100.8384296875,100.783703125],[0.671509376239361,-0.655584233869254,0.241269612064369,-0.247130419452961],[0,0,0,0],[8.999999E+09,8.999999E+09,8.999999E+09,8.999999E+09,8.999999E+09,8.999999E+09]];
	LOCAL CONST Robtarget Tr_meulage_bavure_P210 :=[[-45.33016796875,-104.1663203125,101.6851796875],[0.670476700789359,-0.65630585383525,0.242039737497789,-0.247265819296162],[0,0,0,0],[8.999999E+09,8.999999E+09,8.999999E+09,8.999999E+09,8.999999E+09,8.999999E+09]];
	LOCAL CONST Robtarget Tr_meulage_bavure_P211 :=[[-43.0704609375,-106.147921875,102.213078125],[0.669536368272906,-0.656996936164172,0.242699581721542,-0.247331741721531],[0,0,0,0],[8.999999E+09,8.999999E+09,8.999999E+09,8.999999E+09,8.999999E+09,8.999999E+09]];
	LOCAL CONST Robtarget Tr_meulage_bavure_P212 :=[[-41.735671875,-107.261015625,102.5188125],[0.66874845125707,-0.657695484147894,0.243114062661674,-0.247199740309073],[0,0,0,0],[8.999999E+09,8.999999E+09,8.999999E+09,8.999999E+09,8.999999E+09,8.999999E+09]];
	LOCAL CONST Robtarget Tr_meulage_bavure_P213 :=[[-37.615921875,-110.9701015625,103.4914765625],[0.668154072949221,-0.65839581910775,0.243226701257067,-0.246831626779083],[0,0,0,0],[8.999999E+09,8.999999E+09,8.999999E+09,8.999999E+09,8.999999E+09,8.999999E+09]];
	LOCAL CONST Robtarget Tr_meulage_bavure_P214 :=[[-35.34746484375,-112.9839609375,104.02403125],[0.667738478617938,-0.659051067687565,0.243113713418496,-0.246318364521917],[0,0,0,0],[8.999999E+09,8.999999E+09,8.999999E+09,8.999999E+09,8.999999E+09,8.999999E+09]];
	LOCAL CONST Robtarget Tr_meulage_bavure_P215 :=[[-34.55,-113.696375,104.2117265625],[0.667444766287101,-0.659599543601335,0.242933832718058,-0.245823267730663],[0,0,0,0],[8.999999E+09,8.999999E+09,8.999999E+09,8.999999E+09,8.999999E+09,8.999999E+09]];
	LOCAL CONST Robtarget Tr_meulage_bavure_P216 :=[[-32.82621484375,-115.2352265625,104.6173125],[0.667208230555697,-0.659970030340608,0.242870118751149,-0.245533789016412],[0,0,0,0],[8.999999E+09,8.999999E+09,8.999999E+09,8.999999E+09,8.999999E+09,8.999999E+09]];
	LOCAL CONST Robtarget Tr_meulage_bavure_P217 :=[[-32.04440234375,-115.865,104.79403125],[0.666994225643563,-0.660120535436869,0.24302591119863,-0.245556486655843],[0,0,0,0],[8.999999E+09,8.999999E+09,8.999999E+09,8.999999E+09,8.999999E+09,8.999999E+09]];
	LOCAL CONST Robtarget Tr_meulage_bavure_P218 :=[[-29.99258984375,-117.5891171875,105.265390625],[0.666813332165311,-0.660069236868941,0.243364073101386,-0.245850585741324],[0,0,0,0],[8.999999E+09,8.999999E+09,8.999999E+09,8.999999E+09,8.999999E+09,8.999999E+09]];
	LOCAL CONST Robtarget Tr_meulage_bavure_P219 :=[[-27.409037109375,-119.661578125,105.848453125],[0.666712219734897,-0.659894714383715,0.243721248835849,-0.246239182199942],[0,0,0,0],[8.999999E+09,8.999999E+09,8.999999E+09,8.999999E+09,8.999999E+09,8.999999E+09]];
	LOCAL CONST Robtarget Tr_meulage_bavure_P220 :=[[-26.932634765625,-120.076515625,105.9594453125],[0.666758561225253,-0.659689956206727,0.243885921093987,-0.246499168771284],[0,0,0,0],[8.999999E+09,8.999999E+09,8.999999E+09,8.999999E+09,8.999999E+09,8.999999E+09]];
	LOCAL CONST Robtarget Tr_meulage_bavure_P221 :=[[-26.674736328125,-120.3123125,106.02071875],[0.666992133054392,-0.659525895903362,0.243715660929897,-0.246474671505866],[0,0,0,0],[8.999999E+09,8.999999E+09,8.999999E+09,8.999999E+09,8.999999E+09,8.999999E+09]];
	LOCAL CONST Robtarget Tr_meulage_bavure_P222 :=[[-26.23561328125,-120.69321875,106.122859375],[0.667391405638557,-0.659427223183775,0.243214901942626,-0.246152311540976],[0,0,0,0],[8.999999E+09,8.999999E+09,8.999999E+09,8.999999E+09,8.999999E+09,8.999999E+09]];
	LOCAL CONST Robtarget Tr_meulage_bavure_P223 :=[[-21.49404296875,-124.59453125,107.2033203125],[0.667894964395899,-0.65935964125452,0.242516635935787,-0.245655981636312],[0,0,0,0],[8.999999E+09,8.999999E+09,8.999999E+09,8.999999E+09,8.999999E+09,8.999999E+09]];
	LOCAL CONST Robtarget Tr_meulage_bavure_P224 :=[[-21.286357421875,-124.763234375,107.2504140625],[0.668414395775128,-0.659287084776112,0.24179814774017,-0.245145652862555],[0,0,0,0],[8.999999E+09,8.999999E+09,8.999999E+09,8.999999E+09,8.999999E+09,8.999999E+09]];
	LOCAL CONST Robtarget Tr_meulage_bavure_P225 :=[[-20.704400390625,-125.2962890625,107.38878125],[0.66889091240142,-0.659191287230236,0.241171627357109,-0.244720330795101],[0,0,0,0],[8.999999E+09,8.999999E+09,8.999999E+09,8.999999E+09,8.999999E+09,8.999999E+09]];
	LOCAL CONST Robtarget Tr_meulage_bavure_P226 :=[[-15.6667998046875,-129.8159453125,108.57646875],[0.669310452017579,-0.659092245264467,0.240636171552833,-0.244366863532402],[0,0,0,0],[8.999999E+09,8.999999E+09,8.999999E+09,8.999999E+09,8.999999E+09,8.999999E+09]];
	LOCAL CONST Robtarget Tr_meulage_bavure_P227 :=[[-13.746203125,-131.537765625,109.029140625],[0.669679128534316,-0.659035094361163,0.240130133073073,-0.244008459681629],[0,0,0,0],[8.999999E+09,8.999999E+09,8.999999E+09,8.999999E+09,8.999999E+09,8.999999E+09]];
	LOCAL CONST Robtarget Tr_meulage_bavure_P228 :=[[-11.9880673828125,-133.06496875,109.4383203125],[0.669996870343958,-0.659040981789208,0.239629027431175,-0.243612617210208],[0,0,0,0],[8.999999E+09,8.999999E+09,8.999999E+09,8.999999E+09,8.999999E+09,8.999999E+09]];
	LOCAL CONST Robtarget Tr_meulage_bavure_P229 :=[[-8.7636748046875,-135.768875,110.17846875],[0.670237172267853,-0.659079114111976,0.239210117403008,-0.243259889796498],[0,0,0,0],[8.999999E+09,8.999999E+09,8.999999E+09,8.999999E+09,8.999999E+09,8.999999E+09]];
	LOCAL CONST Robtarget Tr_meulage_bavure_P230 :=[[-2.16247875976563,-141.200796875,111.682734375],[0.670326789084152,-0.659108669355568,0.239035780845299,-0.243104202539038],[0,0,0,0],[8.999999E+09,8.999999E+09,8.999999E+09,8.999999E+09,8.999999E+09,8.999999E+09]];
	LOCAL CONST Robtarget Tr_meulage_bavure_P231 :=[[-1.49243212890625,-141.794015625,111.8398671875],[0.670214014782882,-0.659066461040377,0.239261015294065,-0.243307913724106],[0,0,0,0],[8.999999E+09,8.999999E+09,8.999999E+09,8.999999E+09,8.999999E+09,8.999999E+09]];
	LOCAL CONST Robtarget Tr_meulage_bavure_P232 :=[[1.29419274902344,-144.11309375,112.477640625],[0.669875430708055,-0.658929959893536,0.23994747535837,-0.243933237500642],[0,0,0,0],[8.999999E+09,8.999999E+09,8.999999E+09,8.999999E+09,8.999999E+09,8.999999E+09]];
	LOCAL CONST Robtarget Tr_meulage_bavure_P233 :=[[4.381544921875,-146.861734375,113.2032734375],[0.669325244360453,-0.658727394729108,0.241036792672152,-0.244914681621057],[0,0,0,0],[8.999999E+09,8.999999E+09,8.999999E+09,8.999999E+09,8.999999E+09,8.999999E+09]];
	LOCAL CONST Robtarget Tr_meulage_bavure_P234 :=[[4.754892578125,-147.173515625,113.2888359375],[0.668659687350122,-0.65845824138153,0.242376321217312,-0.246131440053363],[0,0,0,0],[8.999999E+09,8.999999E+09,8.999999E+09,8.999999E+09,8.999999E+09,8.999999E+09]];
	LOCAL CONST Robtarget Tr_meulage_bavure_P235 :=[[5.6457626953125,-147.9608125,113.4976015625],[0.667920831130551,-0.658174203372147,0.243838560929941,-0.247449464660826],[0,0,0,0],[8.999999E+09,8.999999E+09,8.999999E+09,8.999999E+09,8.999999E+09,8.999999E+09]];
	LOCAL CONST Robtarget Tr_meulage_bavure_P236 :=[[7.01516259765625,-149.048609375,113.805515625],[0.667131611968017,-0.657907521051766,0.245350073629173,-0.248789966491085],[0,0,0,0],[8.999999E+09,8.999999E+09,8.999999E+09,8.999999E+09,8.999999E+09,8.999999E+09]];
	LOCAL CONST Robtarget Tr_meulage_bavure_P237 :=[[7.78588330078125,-149.83540625,113.9973359375],[0.666340481522088,-0.657641177113687,0.246855834828783,-0.250121253915816],[0,0,0,0],[8.999999E+09,8.999999E+09,8.999999E+09,8.999999E+09,8.999999E+09,8.999999E+09]];
	LOCAL CONST Robtarget Tr_meulage_bavure_P238 :=[[9.8191484375,-151.726171875,114.4837734375],[0.665566377742362,-0.657379516511131,0.248322474702574,-0.251415028683835],[0,0,0,0],[8.999999E+09,8.999999E+09,8.999999E+09,8.999999E+09,8.999999E+09,8.999999E+09]];
	LOCAL CONST Robtarget Tr_meulage_bavure_P239 :=[[13.07139453125,-154.67859375,115.2542109375],[0.664852307154308,-0.657148829935617,0.249656723503926,-0.252583343463356],[0,0,0,0],[8.999999E+09,8.999999E+09,8.999999E+09,8.999999E+09,8.999999E+09,8.999999E+09]];
	LOCAL CONST Robtarget Tr_meulage_bavure_P240 :=[[14.076822265625,-155.54096875,115.487046875],[0.664265074592214,-0.656986910436248,0.250718628421324,-0.253496113490847],[0,0,0,0],[8.999999E+09,8.999999E+09,8.999999E+09,8.999999E+09,8.999999E+09,8.999999E+09]];
	LOCAL CONST Robtarget Tr_meulage_bavure_P241 :=[[15.09931640625,-156.2198125,115.702796875],[0.663844646454305,-0.656963435308586,0.251374892754738,-0.254007860772152],[0,0,0,0],[8.999999E+09,8.999999E+09,8.999999E+09,8.999999E+09,8.999999E+09,8.999999E+09]];
	LOCAL CONST Robtarget Tr_meulage_bavure_P242 :=[[15.2701650390625,-156.512390625,115.757859375],[0.663632224789659,-0.65711538810448,0.251525911102139,-0.254020379066848],[0,0,0,0],[8.999999E+09,8.999999E+09,8.999999E+09,8.999999E+09,8.999999E+09,8.999999E+09]];
